LIN {X 0,Y 418.278,Z 217.377,A -85,B 0,C 180,E1 -10094.598,E2 -10094.598} C_VEL
LIN {X 0,Y 418.254,Z 217.38,A -85,B 0,C 180,E1 -10097.606,E2 -10097.606} C_VEL
LIN {X 0,Y 418.225,Z 217.388,A -85,B 0,C 180,E1 -10100.665,E2 -10100.665} C_VEL
LIN {X 0,Y 418.244,Z 217.38,A -85,B 0,C 180,E1 -10103.784,E2 -10103.784} C_VEL
LIN {X 0,Y 418.204,Z 217.387,A -85,B 0,C 180,E1 -10107.049,E2 -10107.049} C_VEL
LIN {X 0,Y 418.221,Z 217.39,A -85,B 0,C 180,E1 -10110.274,E2 -10110.274} C_VEL
LIN {X 0,Y 418.215,Z 217.387,A -85,B 0,C 180,E1 -10113.681,E2 -10113.681} C_VEL
LIN {X 0,Y 418.222,Z 217.384,A -85,B 0,C 180,E1 -10117.226,E2 -10117.226} C_VEL
LIN {X 0,Y 418.217,Z 217.389,A -85,B 0,C 180,E1 -10119.686,E2 -10119.686} C_VEL
LIN {X 0,Y 418.211,Z 217.381,A -85,B 0,C 180,E1 -10122.322,E2 -10122.322} C_VEL
LIN {X 0,Y 418.224,Z 217.386,A -85,B 0,C 180,E1 -10125.11,E2 -10125.11} C_VEL
LIN {X 0,Y 418.223,Z 217.388,A -85,B 0,C 180,E1 -10127.767,E2 -10127.767} C_VEL
LIN {X 0,Y 418.231,Z 217.388,A -85,B 0,C 180,E1 -10131.558,E2 -10131.558} C_VEL
LIN {X 0,Y 418.255,Z 217.385,A -85,B 0,C 180,E1 -10135.16,E2 -10135.16} C_VEL
LIN {X 0,Y 418.242,Z 217.388,A -85,B 0,C 180,E1 -10137.473,E2 -10137.473} C_VEL
LIN {X 0,Y 418.296,Z 217.38,A -85,B 0,C 180,E1 -10141.146,E2 -10141.146} C_VEL
LIN {X 0,Y 418.289,Z 217.454,A -85,B 0,C 180,E1 -10141.329,E2 -10141.329} C_VEL
LIN {X 0,Y 421.211,Z 231.065,A -85,B 0,C 180,E1 -10144.291,E2 -10144.291} C_VEL
LIN {X 0,Y 421.805,Z 235.075,A -85,B 0,C 180,E1 -10145.121,E2 -10145.121} C_VEL
LIN {X 0,Y 420.665,Z 251.075,A -85,B 0,C 180,E1 -10148.178,E2 -10148.178} C_VEL
LIN {X 0,Y 419.91,Z 263.661,A -85,B 0,C 180,E1 -10150.553,E2 -10150.553} C_VEL
LIN {X 0,Y 423.793,Z 286.997,A -85,B 0,C 180,E1 -10151.184,E2 -10151.184} C_VEL
LIN {X 0,Y 424.441,Z 292.599,A -85,B 0,C 180,E1 -10151.319,E2 -10151.319} C_VEL
LIN {X 0,Y 423.429,Z 373.284,A -85,B 0,C 180,E1 -10152.741,E2 -10152.741} C_VEL
LIN {X 0,Y 422.9,Z 386.195,A -85,B 0,C 180,E1 -10153.155,E2 -10153.155} C_VEL
LIN {X 0,Y 422.122,Z 398.74,A -85,B 0,C 180,E1 -10153.745,E2 -10153.745} C_VEL
LIN {X 0,Y 421.283,Z 410.718,A -85,B 0,C 180,E1 -10154.519,E2 -10154.519} C_VEL
LIN {X 0,Y 420.456,Z 422.181,A -85,B 0,C 180,E1 -10155.479,E2 -10155.479} C_VEL
LIN {X 0,Y 419.612,Z 432.537,A -85,B 0,C 180,E1 -10156.562,E2 -10156.562} C_VEL
LIN {X 0,Y 419.023,Z 441.025,A -85,B 0,C 180,E1 -10157.652,E2 -10157.652} C_VEL
LIN {X 0,Y 418.225,Z 450.262,A -85,B 0,C 180,E1 -10159.102,E2 -10159.102} C_VEL
LIN {X 0,Y 417.725,Z 457.708,A -85,B 0,C 180,E1 -10160.558,E2 -10160.558} C_VEL
LIN {X 0,Y 417.326,Z 464.595,A -85,B 0,C 180,E1 -10162.256,E2 -10162.256} C_VEL
LIN {X 0,Y 417.128,Z 469.27,A -85,B 0,C 180,E1 -10163.756,E2 -10163.756} C_VEL
LIN {X 0,Y 417.104,Z 472.633,A -85,B 0,C 180,E1 -10165.166,E2 -10165.166} C_VEL
LIN {X 0,Y 417.07,Z 475.706,A -85,B 0,C 180,E1 -10167.101,E2 -10167.101} C_VEL
LIN {X 0,Y 417.091,Z 476.646,A -85,B 0,C 180,E1 -10168.067,E2 -10168.067} C_VEL
LIN {X 0,Y 417.058,Z 477.181,A -85,B 0,C 180,E1 -10169.033,E2 -10169.033} C_VEL
LIN {X 0,Y 417.057,Z 477.284,A -85,B 0,C 180,E1 -10169.998,E2 -10169.998} C_VEL
LIN {X 0,Y 417.091,Z 476.323,A -85,B 0,C 180,E1 -10171.929,E2 -10171.929} C_VEL
LIN {X 0,Y 417.088,Z 475.245,A -85,B 0,C 180,E1 -10172.896,E2 -10172.896} C_VEL
LIN {X 0,Y 417.023,Z 473.703,A -85,B 0,C 180,E1 -10173.863,E2 -10173.863} C_VEL
LIN {X 0,Y 417.13,Z 470.604,A -85,B 0,C 180,E1 -10175.315,E2 -10175.315} C_VEL
LIN {X 0,Y 417.229,Z 466.427,A -85,B 0,C 180,E1 -10176.769,E2 -10176.769} C_VEL
LIN {X 0,Y 417.451,Z 460.038,A -85,B 0,C 180,E1 -10178.469,E2 -10178.469} C_VEL
LIN {X 0,Y 417.799,Z 453.074,A -85,B 0,C 180,E1 -10179.926,E2 -10179.926} C_VEL
LIN {X 0,Y 418.316,Z 444.342,A -85,B 0,C 180,E1 -10181.383,E2 -10181.383} C_VEL
LIN {X 0,Y 418.877,Z 435.383,A -85,B 0,C 180,E1 -10182.596,E2 -10182.596} C_VEL
LIN {X 0,Y 419.619,Z 424.593,A -85,B 0,C 180,E1 -10183.78,E2 -10183.78} C_VEL
LIN {X 0,Y 420.27,Z 413.141,A -85,B 0,C 180,E1 -10184.772,E2 -10184.772} C_VEL
LIN {X 0,Y 421.02,Z 400.592,A -85,B 0,C 180,E1 -10185.612,E2 -10185.612} C_VEL
LIN {X 0,Y 421.634,Z 387.804,A -85,B 0,C 180,E1 -10186.24,E2 -10186.24} C_VEL
LIN {X 0,Y 422.161,Z 374.192,A -85,B 0,C 180,E1 -10186.685,E2 -10186.685} C_VEL
LIN {X 0,Y 422.539,Z 344.069,A -85,B 0,C 180,E1 -10187.23,E2 -10187.23} C_VEL
LIN {X 0,Y 422.928,Z 289.758,A -85,B 0,C 180,E1 -10188.161,E2 -10188.161} C_VEL
LIN {X 0,Y 419.318,Z 264.152,A -85,B 0,C 180,E1 -10188.756,E2 -10188.756} C_VEL
LIN {X 0,Y 420.39,Z 244.757,A -85,B 0,C 180,E1 -10192.35,E2 -10192.35} C_VEL
LIN {X 0,Y 421.057,Z 232.437,A -85,B 0,C 180,E1 -10194.659,E2 -10194.659} C_VEL
LIN {X 0,Y 419.409,Z 222.603,A -85,B 0,C 180,E1 -10196.627,E2 -10196.627} C_VEL
LIN {X 0,Y 418.358,Z 217.376,A -85,B 0,C 180,E1 -10197.726,E2 -10197.726} C_VEL
LIN {X 0,Y 418.196,Z 217.389,A -85,B 0,C 180,E1 -10201.392,E2 -10201.392} C_VEL
LIN {X 0,Y 418.248,Z 217.384,A -85,B 0,C 180,E1 -10204.576,E2 -10204.576} C_VEL
LIN {X 0,Y 418.208,Z 217.393,A -85,B 0,C 180,E1 -10207.829,E2 -10207.829} C_VEL
LIN {X 0,Y 418.199,Z 217.388,A -85,B 0,C 180,E1 -10210.944,E2 -10210.944} C_VEL
LIN {X 0,Y 418.185,Z 217.396,A -85,B 0,C 180,E1 -10213.725,E2 -10213.725} C_VEL
LIN {X 0,Y 418.234,Z 217.385,A -85,B 0,C 180,E1 -10216.451,E2 -10216.451} C_VEL
LIN {X 0,Y 418.238,Z 217.384,A -85,B 0,C 180,E1 -10219.119,E2 -10219.119} C_VEL
LIN {X 0,Y 418.206,Z 217.39,A -85,B 0,C 180,E1 -10222.161,E2 -10222.161} C_VEL
LIN {X 0,Y 418.23,Z 217.389,A -85,B 0,C 180,E1 -10225.416,E2 -10225.416} C_VEL
LIN {X 0,Y 418.177,Z 217.391,A -85,B 0,C 180,E1 -10228.601,E2 -10228.601} C_VEL
LIN {X 0,Y 418.255,Z 217.384,A -85,B 0,C 180,E1 -10231.934,E2 -10231.934} C_VEL
LIN {X 0,Y 418.249,Z 217.385,A -85,B 0,C 180,E1 -10235.16,E2 -10235.16} C_VEL
LIN {X 0,Y 418.218,Z 217.386,A -85,B 0,C 180,E1 -10238.302,E2 -10238.302} C_VEL
LIN {X 0,Y 418.239,Z 217.391,A -85,B 0,C 180,E1 -10241.381,E2 -10241.381} C_VEL
LIN {X 0,Y 418.263,Z 217.38,A -85,B 0,C 180,E1 -10244.404,E2 -10244.404} C_VEL
LIN {X 0,Y 418.323,Z 217.379,A -85,B 0,C 180,E1 -10247.384,E2 -10247.384} C_VEL
LIN {X 0,Y 418.368,Z 217.374,A -85,B 0,C 180,E1 -10251.304,E2 -10251.304} C_VEL
LIN {X 0,Y 418.49,Z 217.352,A -85,B 0,C 180,E1 -10254.217,E2 -10254.217} C_VEL
LIN {X 0,Y 418.492,Z 217.352,A -85,B 0,C 180,E1 -10258.075,E2 -10258.075} C_VEL
LIN {X 0,Y 418.62,Z 217.336,A -85,B 0,C 180,E1 -10260,E2 -10260} C_VEL
LIN {X 0,Y 418.45,Z 217.363,A -85,B 0,C 180,E1 -10262.888,E2 -10262.888} C_VEL
LIN {X 0,Y 418.438,Z 217.363,A -85,B 0,C 180,E1 -10266.752,E2 -10266.752} C_VEL
LIN {X 0,Y 418.294,Z 217.377,A -85,B 0,C 180,E1 -10269.672,E2 -10269.672} C_VEL
LIN {X 0,Y 418.306,Z 217.38,A -85,B 0,C 180,E1 -10273.007,E2 -10273.007} C_VEL
LIN {X 0,Y 418.272,Z 217.386,A -85,B 0,C 180,E1 -10276.74,E2 -10276.74} C_VEL
LIN {X 0,Y 418.223,Z 217.385,A -85,B 0,C 180,E1 -10279.791,E2 -10279.791} C_VEL
LIN {X 0,Y 418.187,Z 217.397,A -85,B 0,C 180,E1 -10282.739,E2 -10282.739} C_VEL
LIN {X 0,Y 418.226,Z 217.385,A -85,B 0,C 180,E1 -10285.907,E2 -10285.907} C_VEL
LIN {X 0,Y 418.223,Z 217.386,A -85,B 0,C 180,E1 -10289.165,E2 -10289.165} C_VEL
LIN {X 0,Y 418.218,Z 217.389,A -85,B 0,C 180,E1 -10292.847,E2 -10292.847} C_VEL
LIN {X 0,Y 418.208,Z 217.392,A -85,B 0,C 180,E1 -10296.241,E2 -10296.241} C_VEL
LIN {X 0,Y 418.208,Z 217.388,A -85,B 0,C 180,E1 -10299.686,E2 -10299.686} C_VEL
LIN {X 0,Y 418.196,Z 217.396,A -85,B 0,C 180,E1 -10302.324,E2 -10302.324} C_VEL
LIN {X 0,Y 418.205,Z 217.388,A -85,B 0,C 180,E1 -10305.112,E2 -10305.112} C_VEL
LIN {X 0,Y 418.212,Z 217.389,A -85,B 0,C 180,E1 -10307.77,E2 -10307.77} C_VEL
LIN {X 0,Y 418.232,Z 217.387,A -85,B 0,C 180,E1 -10310.622,E2 -10310.622} C_VEL
LIN {X 0,Y 418.221,Z 217.391,A -85,B 0,C 180,E1 -10313.98,E2 -10313.98} C_VEL
LIN {X 0,Y 418.238,Z 217.383,A -85,B 0,C 180,E1 -10317.16,E2 -10317.16} C_VEL
LIN {X 0,Y 418.252,Z 217.382,A -85,B 0,C 180,E1 -10320.899,E2 -10320.899} C_VEL
LIN {X 0,Y 418.254,Z 217.387,A -85,B 0,C 180,E1 -10324.099,E2 -10324.099} C_VEL
LIN {X 0,Y 418.22,Z 217.386,A -85,B 0,C 180,E1 -10327.267,E2 -10327.267} C_VEL
LIN {X 0,Y 418.273,Z 217.381,A -85,B 0,C 180,E1 -10330.367,E2 -10330.367} C_VEL
LIN {X 0,Y 418.308,Z 217.377,A -85,B 0,C 180,E1 -10333.408,E2 -10333.408} C_VEL
LIN {X 0,Y 418.34,Z 217.371,A -85,B 0,C 180,E1 -10337.002,E2 -10337.002} C_VEL
LIN {X 0,Y 418.334,Z 217.372,A -85,B 0,C 180,E1 -10340.331,E2 -10340.331} C_VEL
LIN {X 0,Y 418.456,Z 217.363,A -85,B 0,C 180,E1 -10343.251,E2 -10343.251} C_VEL
LIN {X 0,Y 418.477,Z 217.455,A -85,B 0,C 180,E1 -10343.947,E2 -10343.947} C_VEL
LIN {X 0,Y 419.779,Z 226.103,A -85,B 0,C 180,E1 -10345.922,E2 -10345.922} C_VEL
LIN {X 0,Y 419.767,Z 228.219,A -85,B 0,C 180,E1 -10346.357,E2 -10346.357} C_VEL
LIN {X 0,Y 423.446,Z 246.784,A -85,B 0,C 180,E1 -10346.827,E2 -10346.827} C_VEL
LIN {X 0,Y 422.508,Z 326.828,A -85,B 0,C 180,E1 -10348.186,E2 -10348.186} C_VEL
LIN {X 0,Y 421.787,Z 330.749,A -85,B 0,C 180,E1 -10348.232,E2 -10348.232} C_VEL
LIN {X 0,Y 415.99,Z 342.937,A -85,B 0,C 180,E1 -10348.344,E2 -10348.344} C_VEL
LIN {X 0,Y 415.247,Z 346.753,A -85,B 0,C 180,E1 -10348.46,E2 -10348.46} C_VEL
LIN {X 0,Y 414.843,Z 359.25,A -85,B 0,C 180,E1 -10349.031,E2 -10349.031} C_VEL
LIN {X 0,Y 414.324,Z 370.985,A -85,B 0,C 180,E1 -10349.758,E2 -10349.758} C_VEL
LIN {X 0,Y 413.654,Z 381.718,A -85,B 0,C 180,E1 -10350.61,E2 -10350.61} C_VEL
LIN {X 0,Y 412.91,Z 392.654,A -85,B 0,C 180,E1 -10351.708,E2 -10351.708} C_VEL
LIN {X 0,Y 412.267,Z 402.428,A -85,B 0,C 180,E1 -10352.933,E2 -10352.933} C_VEL
LIN {X 0,Y 411.654,Z 410.465,A -85,B 0,C 180,E1 -10354.162,E2 -10354.162} C_VEL
LIN {X 0,Y 411.105,Z 418.344,A -85,B 0,C 180,E1 -10355.642,E2 -10355.642} C_VEL
LIN {X 0,Y 410.777,Z 424.544,A -85,B 0,C 180,E1 -10357.106,E2 -10357.106} C_VEL
LIN {X 0,Y 410.393,Z 430.353,A -85,B 0,C 180,E1 -10358.867,E2 -10358.867} C_VEL
LIN {X 0,Y 410.172,Z 434.052,A -85,B 0,C 180,E1 -10360.365,E2 -10360.365} C_VEL
LIN {X 0,Y 410.037,Z 437.334,A -85,B 0,C 180,E1 -10362.32,E2 -10362.32} C_VEL
LIN {X 0,Y 409.887,Z 438.786,A -85,B 0,C 180,E1 -10363.89,E2 -10363.89} C_VEL
LIN {X 0,Y 409.889,Z 439.171,A -85,B 0,C 180,E1 -10364.904,E2 -10364.904} C_VEL
LIN {X 0,Y 409.922,Z 439.074,A -85,B 0,C 180,E1 -10366.24,E2 -10366.24} C_VEL
LIN {X 0,Y 409.98,Z 437.835,A -85,B 0,C 180,E1 -10367.973,E2 -10367.973} C_VEL
LIN {X 0,Y 410.24,Z 435.587,A -85,B 0,C 180,E1 -10369.572,E2 -10369.572} C_VEL
LIN {X 0,Y 410.472,Z 432.468,A -85,B 0,C 180,E1 -10371.073,E2 -10371.073} C_VEL
LIN {X 0,Y 410.829,Z 427.769,A -85,B 0,C 180,E1 -10372.731,E2 -10372.731} C_VEL
LIN {X 0,Y 411.322,Z 422.338,A -85,B 0,C 180,E1 -10374.209,E2 -10374.209} C_VEL
LIN {X 0,Y 411.979,Z 415.054,A -85,B 0,C 180,E1 -10375.785,E2 -10375.785} C_VEL
LIN {X 0,Y 412.672,Z 407.471,A -85,B 0,C 180,E1 -10377.1,E2 -10377.1} C_VEL
LIN {X 0,Y 413.52,Z 398.148,A -85,B 0,C 180,E1 -10378.415,E2 -10378.415} C_VEL
LIN {X 0,Y 414.375,Z 388.005,A -85,B 0,C 180,E1 -10379.574,E2 -10379.574} C_VEL
LIN {X 0,Y 415.205,Z 377.739,A -85,B 0,C 180,E1 -10380.516,E2 -10380.516} C_VEL
LIN {X 0,Y 415.907,Z 365.838,A -85,B 0,C 180,E1 -10381.376,E2 -10381.376} C_VEL
LIN {X 0,Y 416.547,Z 352.72,A -85,B 0,C 180,E1 -10382.084,E2 -10382.084} C_VEL
LIN {X 0,Y 416.978,Z 339.811,A -85,B 0,C 180,E1 -10382.558,E2 -10382.558} C_VEL
LIN {X 0,Y 417.233,Z 323.651,A -85,B 0,C 180,E1 -10382.902,E2 -10382.902} C_VEL
LIN {X 0,Y 418.307,Z 248.25,A -85,B 0,C 180,E1 -10384.226,E2 -10384.226} C_VEL
LIN {X 0,Y 414.744,Z 232.783,A -85,B 0,C 180,E1 -10384.718,E2 -10384.718} C_VEL
LIN {X 0,Y 413.422,Z 228.606,A -85,B 0,C 180,E1 -10384.897,E2 -10384.897} C_VEL
LIN {X 0,Y 411.214,Z 218.263,A -85,B 0,C 180,E1 -10387.428,E2 -10387.428} C_VEL
LIN {X 0,Y 411.203,Z 218.265,A -85,B 0,C 180,E1 -10390.499,E2 -10390.499} C_VEL
LIN {X 0,Y 411.211,Z 218.265,A -85,B 0,C 180,E1 -10393.126,E2 -10393.126} C_VEL
LIN {X 0,Y 411.227,Z 218.261,A -85,B 0,C 180,E1 -10395.87,E2 -10395.87} C_VEL
LIN {X 0,Y 411.197,Z 218.264,A -85,B 0,C 180,E1 -10399.498,E2 -10399.498} C_VEL
LIN {X 0,Y 411.187,Z 218.265,A -85,B 0,C 180,E1 -10402.026,E2 -10402.026} C_VEL
LIN {X 0,Y 411.188,Z 218.262,A -85,B 0,C 180,E1 -10405.665,E2 -10405.665} C_VEL
LIN {X 0,Y 411.177,Z 218.262,A -85,B 0,C 180,E1 -10409.152,E2 -10409.152} C_VEL
LIN {X 0,Y 411.24,Z 218.255,A -85,B 0,C 180,E1 -10412.521,E2 -10412.521} C_VEL
LIN {X 0,Y 411.207,Z 218.259,A -85,B 0,C 180,E1 -10415.784,E2 -10415.784} C_VEL
LIN {X 0,Y 411.196,Z 218.256,A -85,B 0,C 180,E1 -10418.966,E2 -10418.966} C_VEL
LIN {X 0,Y 411.229,Z 218.255,A -85,B 0,C 180,E1 -10422.084,E2 -10422.084} C_VEL
LIN {X 0,Y 411.238,Z 218.258,A -85,B 0,C 180,E1 -10425.147,E2 -10425.147} C_VEL
LIN {X 0,Y 411.257,Z 218.253,A -85,B 0,C 180,E1 -10428.167,E2 -10428.167} C_VEL
LIN {X 0,Y 411.419,Z 218.228,A -85,B 0,C 180,E1 -10432.186,E2 -10432.186} C_VEL
LIN {X 0,Y 411.452,Z 218.229,A -85,B 0,C 180,E1 -10434.118,E2 -10434.118} C_VEL
LIN {X 0,Y 411.481,Z 218.223,A -85,B 0,C 180,E1 -10438.043,E2 -10438.043} C_VEL
LIN {X 0,Y 411.611,Z 218.205,A -85,B 0,C 180,E1 -10440,E2 -10440} C_VEL
LIN {X 0,Y 411.428,Z 218.231,A -85,B 0,C 180,E1 -10442.938,E2 -10442.938} C_VEL
LIN {X 0,Y 411.404,Z 218.231,A -85,B 0,C 180,E1 -10446.868,E2 -10446.868} C_VEL
LIN {X 0,Y 411.269,Z 218.244,A -85,B 0,C 180,E1 -10449.84,E2 -10449.84} C_VEL
LIN {X 0,Y 411.289,Z 218.25,A -85,B 0,C 180,E1 -10453.109,E2 -10453.109} C_VEL
LIN {X 0,Y 411.245,Z 218.26,A -85,B 0,C 180,E1 -10456.89,E2 -10456.89} C_VEL
LIN {X 0,Y 411.188,Z 218.259,A -85,B 0,C 180,E1 -10459.989,E2 -10459.989} C_VEL
LIN {X 0,Y 411.17,Z 218.263,A -85,B 0,C 180,E1 -10463.15,E2 -10463.15} C_VEL
LIN {X 0,Y 411.166,Z 218.269,A -85,B 0,C 180,E1 -10466.386,E2 -10466.386} C_VEL
LIN {X 0,Y 411.178,Z 218.264,A -85,B 0,C 180,E1 -10469.715,E2 -10469.715} C_VEL
LIN {X 0,Y 411.188,Z 218.263,A -85,B 0,C 180,E1 -10473.158,E2 -10473.158} C_VEL
LIN {X 0,Y 411.176,Z 218.268,A -85,B 0,C 180,E1 -10476.554,E2 -10476.554} C_VEL
LIN {X 0,Y 411.184,Z 218.265,A -85,B 0,C 180,E1 -10479.726,E2 -10479.726} C_VEL
LIN {X 0,Y 411.159,Z 218.266,A -85,B 0,C 180,E1 -10483.136,E2 -10483.136} C_VEL
LIN {X 0,Y 411.157,Z 218.269,A -85,B 0,C 180,E1 -10485.883,E2 -10485.883} C_VEL
LIN {X 0,Y 411.144,Z 218.269,A -85,B 0,C 180,E1 -10488.775,E2 -10488.775} C_VEL
LIN {X 0,Y 411.18,Z 218.27,A -85,B 0,C 180,E1 -10492.027,E2 -10492.027} C_VEL
LIN {X 0,Y 411.202,Z 218.263,A -85,B 0,C 180,E1 -10495.668,E2 -10495.668} C_VEL
LIN {X 0,Y 411.187,Z 218.267,A -85,B 0,C 180,E1 -10499.153,E2 -10499.153} C_VEL
LIN {X 0,Y 411.245,Z 218.386,A -85,B 0,C 180,E1 -10500.991,E2 -10500.991} C_VEL
LIN {X 0,Y 414.024,Z 231.041,A -85,B 0,C 180,E1 -10503.811,E2 -10503.811} C_VEL
LIN {X 0,Y 414.931,Z 236.363,A -85,B 0,C 180,E1 -10504.948,E2 -10504.948} C_VEL
LIN {X 0,Y 413.75,Z 252.357,A -85,B 0,C 180,E1 -10508.057,E2 -10508.057} C_VEL
LIN {X 0,Y 413.073,Z 263.481,A -85,B 0,C 180,E1 -10510.165,E2 -10510.165} C_VEL
LIN {X 0,Y 417.131,Z 287.273,A -85,B 0,C 180,E1 -10510.834,E2 -10510.834} C_VEL
LIN {X 0,Y 417.841,Z 294.938,A -85,B 0,C 180,E1 -10511.012,E2 -10511.012} C_VEL
LIN {X 0,Y 416.762,Z 372.395,A -85,B 0,C 180,E1 -10512.393,E2 -10512.393} C_VEL
LIN {X 0,Y 416.204,Z 385.488,A -85,B 0,C 180,E1 -10512.812,E2 -10512.812} C_VEL
LIN {X 0,Y 415.417,Z 398.126,A -85,B 0,C 180,E1 -10513.412,E2 -10513.412} C_VEL
LIN {X 0,Y 414.576,Z 409.396,A -85,B 0,C 180,E1 -10514.136,E2 -10514.136} C_VEL
LIN {X 0,Y 413.676,Z 421.043,A -85,B 0,C 180,E1 -10515.11,E2 -10515.11} C_VEL
LIN {X 0,Y 412.805,Z 431.536,A -85,B 0,C 180,E1 -10516.21,E2 -10516.21} C_VEL
LIN {X 0,Y 412.073,Z 441.02,A -85,B 0,C 180,E1 -10517.44,E2 -10517.44} C_VEL
LIN {X 0,Y 411.243,Z 450.174,A -85,B 0,C 180,E1 -10518.915,E2 -10518.915} C_VEL
LIN {X 0,Y 410.699,Z 457.569,A -85,B 0,C 180,E1 -10520.395,E2 -10520.395} C_VEL
LIN {X 0,Y 410.268,Z 464.398,A -85,B 0,C 180,E1 -10522.122,E2 -10522.122} C_VEL
LIN {X 0,Y 410.044,Z 469.361,A -85,B 0,C 180,E1 -10523.775,E2 -10523.775} C_VEL
LIN {X 0,Y 410.011,Z 472.377,A -85,B 0,C 180,E1 -10525.082,E2 -10525.082} C_VEL
LIN {X 0,Y 409.967,Z 475.422,A -85,B 0,C 180,E1 -10527.051,E2 -10527.051} C_VEL
LIN {X 0,Y 410.018,Z 476.351,A -85,B 0,C 180,E1 -10528.034,E2 -10528.034} C_VEL
LIN {X 0,Y 409.981,Z 476.862,A -85,B 0,C 180,E1 -10529.016,E2 -10529.016} C_VEL
LIN {X 0,Y 409.976,Z 476.95,A -85,B 0,C 180,E1 -10529.998,E2 -10529.998} C_VEL
LIN {X 0,Y 410.019,Z 475.965,A -85,B 0,C 180,E1 -10531.963,E2 -10531.963} C_VEL
LIN {X 0,Y 409.987,Z 474.861,A -85,B 0,C 180,E1 -10532.946,E2 -10532.946} C_VEL
LIN {X 0,Y 409.942,Z 473.303,A -85,B 0,C 180,E1 -10533.93,E2 -10533.93} C_VEL
LIN {X 0,Y 410.025,Z 470.174,A -85,B 0,C 180,E1 -10535.407,E2 -10535.407} C_VEL
LIN {X 0,Y 410.16,Z 465.968,A -85,B 0,C 180,E1 -10536.886,E2 -10536.886} C_VEL
LIN {X 0,Y 410.378,Z 459.543,A -85,B 0,C 180,E1 -10538.616,E2 -10538.616} C_VEL
LIN {X 0,Y 410.737,Z 452.536,A -85,B 0,C 180,E1 -10540.098,E2 -10540.098} C_VEL
LIN {X 0,Y 411.306,Z 443.743,A -85,B 0,C 180,E1 -10541.579,E2 -10541.579} C_VEL
LIN {X 0,Y 411.921,Z 434.723,A -85,B 0,C 180,E1 -10542.812,E2 -10542.812} C_VEL
LIN {X 0,Y 412.602,Z 424.803,A -85,B 0,C 180,E1 -10543.919,E2 -10543.919} C_VEL
LIN {X 0,Y 413.277,Z 413.842,A -85,B 0,C 180,E1 -10544.901,E2 -10544.901} C_VEL
LIN {X 0,Y 414.015,Z 401.537,A -85,B 0,C 180,E1 -10545.756,E2 -10545.756} C_VEL
LIN {X 0,Y 414.68,Z 388.616,A -85,B 0,C 180,E1 -10546.425,E2 -10546.425} C_VEL
LIN {X 0,Y 415.212,Z 375.583,A -85,B 0,C 180,E1 -10546.878,E2 -10546.878} C_VEL
LIN {X 0,Y 415.506,Z 358.931,A -85,B 0,C 180,E1 -10547.214,E2 -10547.214} C_VEL
LIN {X 0,Y 416.104,Z 290.614,A -85,B 0,C 180,E1 -10548.4,E2 -10548.4} C_VEL
LIN {X 0,Y 412.373,Z 263.746,A -85,B 0,C 180,E1 -10549.051,E2 -10549.051} C_VEL
LIN {X 0,Y 413.58,Z 242.792,A -85,B 0,C 180,E1 -10553.003,E2 -10553.003} C_VEL
LIN {X 0,Y 414.076,Z 233.186,A -85,B 0,C 180,E1 -10554.835,E2 -10554.835} C_VEL
LIN {X 0,Y 411.933,Z 221.274,A -85,B 0,C 180,E1 -10557.277,E2 -10557.277} C_VEL
LIN {X 0,Y 411.296,Z 218.257,A -85,B 0,C 180,E1 -10557.954,E2 -10557.954} C_VEL
LIN {X 0,Y 411.168,Z 218.264,A -85,B 0,C 180,E1 -10561.279,E2 -10561.279} C_VEL
LIN {X 0,Y 411.189,Z 218.265,A -85,B 0,C 180,E1 -10564.329,E2 -10564.329} C_VEL
LIN {X 0,Y 411.174,Z 218.271,A -85,B 0,C 180,E1 -10567.97,E2 -10567.97} C_VEL
LIN {X 0,Y 411.14,Z 218.268,A -85,B 0,C 180,E1 -10571.224,E2 -10571.224} C_VEL
LIN {X 0,Y 411.155,Z 218.267,A -85,B 0,C 180,E1 -10574.486,E2 -10574.486} C_VEL
LIN {X 0,Y 411.199,Z 218.262,A -85,B 0,C 180,E1 -10577.293,E2 -10577.293} C_VEL
LIN {X 0,Y 411.201,Z 218.26,A -85,B 0,C 180,E1 -10580.774,E2 -10580.774} C_VEL
LIN {X 0,Y 411.165,Z 218.265,A -85,B 0,C 180,E1 -10584.468,E2 -10584.468} C_VEL
LIN {X 0,Y 411.172,Z 218.264,A -85,B 0,C 180,E1 -10586.87,E2 -10586.87} C_VEL
LIN {X 0,Y 411.201,Z 218.26,A -85,B 0,C 180,E1 -10590.639,E2 -10590.639} C_VEL
LIN {X 0,Y 411.199,Z 218.266,A -85,B 0,C 180,E1 -10593.616,E2 -10593.616} C_VEL
LIN {X 0,Y 411.214,Z 218.264,A -85,B 0,C 180,E1 -10597.337,E2 -10597.337} C_VEL
LIN {X 0,Y 411.222,Z 218.258,A -85,B 0,C 180,E1 -10600.029,E2 -10600.029} C_VEL
LIN {X 0,Y 411.219,Z 218.262,A -85,B 0,C 180,E1 -10603.129,E2 -10603.129} C_VEL
LIN {X 0,Y 411.266,Z 218.254,A -85,B 0,C 180,E1 -10606.89,E2 -10606.89} C_VEL
LIN {X 0,Y 411.265,Z 218.252,A -85,B 0,C 180,E1 -10610.16,E2 -10610.16} C_VEL
LIN {X 0,Y 411.429,Z 218.238,A -85,B 0,C 180,E1 -10613.132,E2 -10613.132} C_VEL
LIN {X 0,Y 411.268,Z 218.258,A -85,B 0,C 180,E1 -10615.098,E2 -10615.098} C_VEL
LIN {X 0,Y 411.461,Z 218.228,A -85,B 0,C 180,E1 -10618.042,E2 -10618.042} C_VEL
LIN {X 0,Y 411.59,Z 218.212,A -85,B 0,C 180,E1 -10620,E2 -10620} C_VEL
LIN {X 0,Y 411.407,Z 218.241,A -85,B 0,C 180,E1 -10622.937,E2 -10622.937} C_VEL
LIN {X 0,Y 411.402,Z 218.241,A -85,B 0,C 180,E1 -10626.868,E2 -10626.868} C_VEL
LIN {X 0,Y 411.247,Z 218.254,A -85,B 0,C 180,E1 -10629.84,E2 -10629.84} C_VEL
LIN {X 0,Y 411.265,Z 218.256,A -85,B 0,C 180,E1 -10633.109,E2 -10633.109} C_VEL
LIN {X 0,Y 411.215,Z 218.264,A -85,B 0,C 180,E1 -10636.89,E2 -10636.89} C_VEL
LIN {X 0,Y 411.164,Z 218.265,A -85,B 0,C 180,E1 -10639.99,E2 -10639.99} C_VEL
LIN {X 0,Y 411.152,Z 218.268,A -85,B 0,C 180,E1 -10643.15,E2 -10643.15} C_VEL
LIN {X 0,Y 411.195,Z 218.265,A -85,B 0,C 180,E1 -10646.384,E2 -10646.384} C_VEL
LIN {X 0,Y 411.159,Z 218.265,A -85,B 0,C 180,E1 -10649.716,E2 -10649.716} C_VEL
LIN {X 0,Y 411.168,Z 218.265,A -85,B 0,C 180,E1 -10653.159,E2 -10653.159} C_VEL
LIN {X 0,Y 411.156,Z 218.272,A -85,B 0,C 180,E1 -10656.556,E2 -10656.556} C_VEL
LIN {X 0,Y 411.173,Z 218.264,A -85,B 0,C 180,E1 -10659.73,E2 -10659.73} C_VEL
LIN {X 0,Y 411.141,Z 218.268,A -85,B 0,C 180,E1 -10663.137,E2 -10663.137} C_VEL
LIN {X 0,Y 411.139,Z 218.27,A -85,B 0,C 180,E1 -10665.885,E2 -10665.885} C_VEL
LIN {X 0,Y 411.138,Z 218.269,A -85,B 0,C 180,E1 -10668.775,E2 -10668.775} C_VEL
LIN {X 0,Y 411.182,Z 218.265,A -85,B 0,C 180,E1 -10671.835,E2 -10671.835} C_VEL
LIN {X 0,Y 411.19,Z 218.261,A -85,B 0,C 180,E1 -10675.125,E2 -10675.125} C_VEL
LIN {X 0,Y 411.146,Z 218.273,A -85,B 0,C 180,E1 -10678.006,E2 -10678.006} C_VEL
LIN {X 0,Y 411.201,Z 218.261,A -85,B 0,C 180,E1 -10681.414,E2 -10681.414} C_VEL
LIN {X 0,Y 411.222,Z 218.26,A -85,B 0,C 180,E1 -10683.623,E2 -10683.623} C_VEL
LIN {X 0,Y 411.183,Z 218.262,A -85,B 0,C 180,E1 -10686.855,E2 -10686.855} C_VEL
LIN {X 0,Y 411.204,Z 218.265,A -85,B 0,C 180,E1 -10690.054,E2 -10690.054} C_VEL
LIN {X 0,Y 411.255,Z 218.254,A -85,B 0,C 180,E1 -10693.134,E2 -10693.134} C_VEL
LIN {X 0,Y 411.299,Z 218.248,A -85,B 0,C 180,E1 -10696.899,E2 -10696.899} C_VEL
LIN {X 0,Y 411.286,Z 218.252,A -85,B 0,C 180,E1 -10700.164,E2 -10700.164} C_VEL
LIN {X 0,Y 411.42,Z 218.239,A -85,B 0,C 180,E1 -10703.135,E2 -10703.135} C_VEL
LIN {X 0,Y 411.42,Z 218.273,A -85,B 0,C 180,E1 -10703.75,E2 -10703.75} C_VEL
LIN {X 0,Y 412.817,Z 227.357,A -85,B 0,C 180,E1 -10705.853,E2 -10705.853} C_VEL
LIN {X 0,Y 412.784,Z 228.329,A -85,B 0,C 180,E1 -10706.066,E2 -10706.066} C_VEL
LIN {X 0,Y 416.633,Z 248.07,A -85,B 0,C 180,E1 -10706.584,E2 -10706.584} C_VEL
LIN {X 0,Y 415.517,Z 335.676,A -85,B 0,C 180,E1 -10708.117,E2 -10708.117} C_VEL
LIN {X 0,Y 415.247,Z 346.753,A -85,B 0,C 180,E1 -10708.46,E2 -10708.46} C_VEL
LIN {X 0,Y 414.791,Z 350.532,A -85,B 0,C 180,E1 -10708.599,E2 -10708.599} C_VEL
LIN {X 0,Y 412.675,Z 357.887,A -85,B 0,C 180,E1 -10708.878,E2 -10708.878} C_VEL
LIN {X 0,Y 408.624,Z 368.519,A -85,B 0,C 180,E1 -10709.384,E2 -10709.384} C_VEL
LIN {X 0,Y 407.341,Z 373.768,A -85,B 0,C 180,E1 -10709.725,E2 -10709.725} C_VEL
LIN {X 0,Y 407.152,Z 375.467,A -85,B 0,C 180,E1 -10709.856,E2 -10709.856} C_VEL
LIN {X 0,Y 406.374,Z 386.883,A -85,B 0,C 180,E1 -10710.869,E2 -10710.869} C_VEL
LIN {X 0,Y 405.664,Z 396.876,A -85,B 0,C 180,E1 -10711.987,E2 -10711.987} C_VEL
LIN {X 0,Y 405.016,Z 405.922,A -85,B 0,C 180,E1 -10713.234,E2 -10713.234} C_VEL
LIN {X 0,Y 404.404,Z 414.749,A -85,B 0,C 180,E1 -10714.736,E2 -10714.736} C_VEL
LIN {X 0,Y 403.901,Z 421.836,A -85,B 0,C 180,E1 -10716.245,E2 -10716.245} C_VEL
LIN {X 0,Y 403.479,Z 428.302,A -85,B 0,C 180,E1 -10718.011,E2 -10718.011} C_VEL
LIN {X 0,Y 403.189,Z 432.576,A -85,B 0,C 180,E1 -10719.533,E2 -10719.533} C_VEL
LIN {X 0,Y 403.035,Z 435.77,A -85,B 0,C 180,E1 -10721.059,E2 -10721.059} C_VEL
LIN {X 0,Y 402.939,Z 437.731,A -85,B 0,C 180,E1 -10722.383,E2 -10722.383} C_VEL
LIN {X 0,Y 402.804,Z 439.221,A -85,B 0,C 180,E1 -10724.139,E2 -10724.139} C_VEL
LIN {X 0,Y 402.806,Z 439.538,A -85,B 0,C 180,E1 -10725.172,E2 -10725.172} C_VEL
LIN {X 0,Y 402.837,Z 439.382,A -85,B 0,C 180,E1 -10726.354,E2 -10726.354} C_VEL
LIN {X 0,Y 402.933,Z 437.916,A -85,B 0,C 180,E1 -10728.298,E2 -10728.298} C_VEL
LIN {X 0,Y 403.181,Z 435.861,A -85,B 0,C 180,E1 -10729.731,E2 -10729.731} C_VEL
LIN {X 0,Y 403.468,Z 432.239,A -85,B 0,C 180,E1 -10731.457,E2 -10731.457} C_VEL
LIN {X 0,Y 403.893,Z 427.568,A -85,B 0,C 180,E1 -10733.08,E2 -10733.08} C_VEL
LIN {X 0,Y 404.439,Z 421.741,A -85,B 0,C 180,E1 -10734.648,E2 -10734.648} C_VEL
LIN {X 0,Y 405.197,Z 414.151,A -85,B 0,C 180,E1 -10736.249,E2 -10736.249} C_VEL
LIN {X 0,Y 405.944,Z 406.31,A -85,B 0,C 180,E1 -10737.588,E2 -10737.588} C_VEL
LIN {X 0,Y 406.815,Z 396.685,A -85,B 0,C 180,E1 -10738.928,E2 -10738.928} C_VEL
LIN {X 0,Y 407.671,Z 387.16,A -85,B 0,C 180,E1 -10739.995,E2 -10739.995} C_VEL
LIN {X 0,Y 408.631,Z 375.193,A -85,B 0,C 180,E1 -10741.061,E2 -10741.061} C_VEL
LIN {X 0,Y 409.391,Z 363.647,A -85,B 0,C 180,E1 -10741.861,E2 -10741.861} C_VEL
LIN {X 0,Y 409.966,Z 351.271,A -85,B 0,C 180,E1 -10742.501,E2 -10742.501} C_VEL
LIN {X 0,Y 410.355,Z 337.734,A -85,B 0,C 180,E1 -10742.975,E2 -10742.975} C_VEL
LIN {X 0,Y 410.996,Z 299.806,A -85,B 0,C 180,E1 -10743.684,E2 -10743.684} C_VEL
LIN {X 0,Y 411.835,Z 249.631,A -85,B 0,C 180,E1 -10744.574,E2 -10744.574} C_VEL
LIN {X 0,Y 408.153,Z 234.005,A -85,B 0,C 180,E1 -10745.089,E2 -10745.089} C_VEL
LIN {X 0,Y 406.263,Z 228.932,A -85,B 0,C 180,E1 -10745.328,E2 -10745.328} C_VEL
LIN {X 0,Y 404.145,Z 219.145,A -85,B 0,C 180,E1 -10747.804,E2 -10747.804} C_VEL
LIN {X 0,Y 404.154,Z 219.137,A -85,B 0,C 180,E1 -10751.358,E2 -10751.358} C_VEL
LIN {X 0,Y 404.186,Z 219.142,A -85,B 0,C 180,E1 -10754.528,E2 -10754.528} C_VEL
LIN {X 0,Y 404.197,Z 219.135,A -85,B 0,C 180,E1 -10757.304,E2 -10757.304} C_VEL
LIN {X 0,Y 404.155,Z 219.141,A -85,B 0,C 180,E1 -10759.954,E2 -10759.954} C_VEL
LIN {X 0,Y 404.124,Z 219.142,A -85,B 0,C 180,E1 -10763.123,E2 -10763.123} C_VEL
LIN {X 0,Y 404.127,Z 219.147,A -85,B 0,C 180,E1 -10766.186,E2 -10766.186} C_VEL
LIN {X 0,Y 404.133,Z 219.144,A -85,B 0,C 180,E1 -10769.714,E2 -10769.714} C_VEL
LIN {X 0,Y 404.175,Z 219.135,A -85,B 0,C 180,E1 -10773.122,E2 -10773.122} C_VEL
LIN {X 0,Y 404.151,Z 219.139,A -85,B 0,C 180,E1 -10776.425,E2 -10776.425} C_VEL
LIN {X 0,Y 404.184,Z 219.136,A -85,B 0,C 180,E1 -10779.868,E2 -10779.868} C_VEL
LIN {X 0,Y 404.195,Z 219.13,A -85,B 0,C 180,E1 -10782.992,E2 -10782.992} C_VEL
LIN {X 0,Y 404.259,Z 219.125,A -85,B 0,C 180,E1 -10786.938,E2 -10786.938} C_VEL
LIN {X 0,Y 404.232,Z 219.13,A -85,B 0,C 180,E1 -10789.988,E2 -10789.988} C_VEL
LIN {X 0,Y 404.384,Z 219.107,A -85,B 0,C 180,E1 -10793.013,E2 -10793.013} C_VEL
LIN {X 0,Y 404.257,Z 219.128,A -85,B 0,C 180,E1 -10795.014,E2 -10795.014} C_VEL
LIN {X 0,Y 404.451,Z 219.099,A -85,B 0,C 180,E1 -10798.009,E2 -10798.009} C_VEL
LIN {X 0,Y 404.581,Z 219.08,A -85,B 0,C 180,E1 -10800,E2 -10800} C_VEL
LIN {X 0,Y 404.386,Z 219.109,A -85,B 0,C 180,E1 -10802.989,E2 -10802.989} C_VEL
LIN {X 0,Y 404.355,Z 219.11,A -85,B 0,C 180,E1 -10806.989,E2 -10806.989} C_VEL
LIN {X 0,Y 404.237,Z 219.124,A -85,B 0,C 180,E1 -10811.026,E2 -10811.026} C_VEL
LIN {X 0,Y 404.187,Z 219.13,A -85,B 0,C 180,E1 -10814.089,E2 -10814.089} C_VEL
LIN {X 0,Y 404.184,Z 219.136,A -85,B 0,C 180,E1 -10817.194,E2 -10817.194} C_VEL
LIN {X 0,Y 404.134,Z 219.14,A -85,B 0,C 180,E1 -10820.353,E2 -10820.353} C_VEL
LIN {X 0,Y 404.132,Z 219.138,A -85,B 0,C 180,E1 -10823.577,E2 -10823.577} C_VEL
LIN {X 0,Y 404.109,Z 219.143,A -85,B 0,C 180,E1 -10826.884,E2 -10826.884} C_VEL
LIN {X 0,Y 404.125,Z 219.146,A -85,B 0,C 180,E1 -10830.287,E2 -10830.287} C_VEL
LIN {X 0,Y 404.122,Z 219.143,A -85,B 0,C 180,E1 -10833.815,E2 -10833.815} C_VEL
LIN {X 0,Y 404.119,Z 219.143,A -85,B 0,C 180,E1 -10836.876,E2 -10836.876} C_VEL
LIN {X 0,Y 404.137,Z 219.144,A -85,B 0,C 180,E1 -10840.082,E2 -10840.082} C_VEL
LIN {X 0,Y 404.139,Z 219.141,A -85,B 0,C 180,E1 -10843.085,E2 -10843.085} C_VEL
LIN {X 0,Y 404.138,Z 219.143,A -85,B 0,C 180,E1 -10845.927,E2 -10845.927} C_VEL
LIN {X 0,Y 404.1,Z 219.148,A -85,B 0,C 180,E1 -10848.635,E2 -10848.635} C_VEL
LIN {X 0,Y 404.134,Z 219.144,A -85,B 0,C 180,E1 -10851.496,E2 -10851.496} C_VEL
LIN {X 0,Y 404.18,Z 219.139,A -85,B 0,C 180,E1 -10854.985,E2 -10854.985} C_VEL
LIN {X 0,Y 404.139,Z 219.145,A -85,B 0,C 180,E1 -10858.555,E2 -10858.555} C_VEL
LIN {X 0,Y 404.196,Z 219.213,A -85,B 0,C 180,E1 -10860.612,E2 -10860.612} C_VEL
LIN {X 0,Y 406.836,Z 231.026,A -85,B 0,C 180,E1 -10863.312,E2 -10863.312} C_VEL
LIN {X 0,Y 408.047,Z 237.678,A -85,B 0,C 180,E1 -10864.769,E2 -10864.769} C_VEL
LIN {X 0,Y 406.84,Z 253.642,A -85,B 0,C 180,E1 -10867.931,E2 -10867.931} C_VEL
LIN {X 0,Y 406.199,Z 263.14,A -85,B 0,C 180,E1 -10869.755,E2 -10869.755} C_VEL
LIN {X 0,Y 409.938,Z 284.035,A -85,B 0,C 180,E1 -10870.369,E2 -10870.369} C_VEL
LIN {X 0,Y 411.262,Z 294.737,A -85,B 0,C 180,E1 -10870.644,E2 -10870.644} C_VEL
LIN {X 0,Y 410.141,Z 371.606,A -85,B 0,C 180,E1 -10872.035,E2 -10872.035} C_VEL
LIN {X 0,Y 409.623,Z 384.077,A -85,B 0,C 180,E1 -10872.431,E2 -10872.431} C_VEL
LIN {X 0,Y 408.84,Z 396.418,A -85,B 0,C 180,E1 -10873.008,E2 -10873.008} C_VEL
LIN {X 0,Y 407.902,Z 408.004,A -85,B 0,C 180,E1 -10873.741,E2 -10873.741} C_VEL
LIN {X 0,Y 406.919,Z 419.905,A -85,B 0,C 180,E1 -10874.729,E2 -10874.729} C_VEL
LIN {X 0,Y 406.005,Z 430.472,A -85,B 0,C 180,E1 -10875.839,E2 -10875.839} C_VEL
LIN {X 0,Y 405.135,Z 441.004,A -85,B 0,C 180,E1 -10877.221,E2 -10877.221} C_VEL
LIN {X 0,Y 404.257,Z 450.096,A -85,B 0,C 180,E1 -10878.721,E2 -10878.721} C_VEL
LIN {X 0,Y 403.664,Z 457.447,A -85,B 0,C 180,E1 -10880.226,E2 -10880.226} C_VEL
LIN {X 0,Y 403.204,Z 464.218,A -85,B 0,C 180,E1 -10881.983,E2 -10881.983} C_VEL
LIN {X 0,Y 402.935,Z 469.55,A -85,B 0,C 180,E1 -10883.826,E2 -10883.826} C_VEL
LIN {X 0,Y 402.92,Z 472.128,A -85,B 0,C 180,E1 -10884.995,E2 -10884.995} C_VEL
LIN {X 0,Y 402.865,Z 475.142,A -85,B 0,C 180,E1 -10886.999,E2 -10886.999} C_VEL
LIN {X 0,Y 402.946,Z 476.058,A -85,B 0,C 180,E1 -10887.999,E2 -10887.999} C_VEL
LIN {X 0,Y 402.906,Z 476.541,A -85,B 0,C 180,E1 -10888.999,E2 -10888.999} C_VEL
LIN {X 0,Y 402.899,Z 476.616,A -85,B 0,C 180,E1 -10889.998,E2 -10889.998} C_VEL
LIN {X 0,Y 402.948,Z 475.604,A -85,B 0,C 180,E1 -10891.997,E2 -10891.997} C_VEL
LIN {X 0,Y 402.887,Z 474.47,A -85,B 0,C 180,E1 -10892.998,E2 -10892.998} C_VEL
LIN {X 0,Y 402.863,Z 472.898,A -85,B 0,C 180,E1 -10893.999,E2 -10893.999} C_VEL
LIN {X 0,Y 402.922,Z 469.735,A -85,B 0,C 180,E1 -10895.503,E2 -10895.503} C_VEL
LIN {X 0,Y 403.071,Z 465.493,A -85,B 0,C 180,E1 -10897.008,E2 -10897.008} C_VEL
LIN {X 0,Y 403.327,Z 459.029,A -85,B 0,C 180,E1 -10898.767,E2 -10898.767} C_VEL
LIN {X 0,Y 403.69,Z 451.959,A -85,B 0,C 180,E1 -10900.277,E2 -10900.277} C_VEL
LIN {X 0,Y 404.319,Z 443.099,A -85,B 0,C 180,E1 -10901.782,E2 -10901.782} C_VEL
LIN {X 0,Y 404.975,Z 434.017,A -85,B 0,C 180,E1 -10903.035,E2 -10903.035} C_VEL
LIN {X 0,Y 405.686,Z 424.017,A -85,B 0,C 180,E1 -10904.161,E2 -10904.161} C_VEL
LIN {X 0,Y 406.33,Z 412.891,A -85,B 0,C 180,E1 -10905.162,E2 -10905.162} C_VEL
LIN {X 0,Y 407.138,Z 400.433,A -85,B 0,C 180,E1 -10906.03,E2 -10906.03} C_VEL
LIN {X 0,Y 407.781,Z 388.601,A -85,B 0,C 180,E1 -10906.647,E2 -10906.647} C_VEL
LIN {X 0,Y 408.316,Z 375.767,A -85,B 0,C 180,E1 -10907.107,E2 -10907.107} C_VEL
LIN {X 0,Y 408.644,Z 359.413,A -85,B 0,C 180,E1 -10907.448,E2 -10907.448} C_VEL
LIN {X 0,Y 409.283,Z 291.586,A -85,B 0,C 180,E1 -10908.645,E2 -10908.645} C_VEL
LIN {X 0,Y 405.39,Z 263.562,A -85,B 0,C 180,E1 -10909.31,E2 -10909.31} C_VEL
LIN {X 0,Y 406.598,Z 243.538,A -85,B 0,C 180,E1 -10913.152,E2 -10913.152} C_VEL
LIN {X 0,Y 407.1,Z 235.311,A -85,B 0,C 180,E1 -10914.745,E2 -10914.745} C_VEL
LIN {X 0,Y 405.996,Z 227.923,A -85,B 0,C 180,E1 -10916.265,E2 -10916.265} C_VEL
LIN {X 0,Y 404.249,Z 219.134,A -85,B 0,C 180,E1 -10918.132,E2 -10918.132} C_VEL
LIN {X 0,Y 404.124,Z 219.143,A -85,B 0,C 180,E1 -10921.554,E2 -10921.554} C_VEL
LIN {X 0,Y 404.167,Z 219.136,A -85,B 0,C 180,E1 -10925.012,E2 -10925.012} C_VEL
LIN {X 0,Y 404.133,Z 219.141,A -85,B 0,C 180,E1 -10928.753,E2 -10928.753} C_VEL
LIN {X 0,Y 404.099,Z 219.148,A -85,B 0,C 180,E1 -10931.595,E2 -10931.595} C_VEL
LIN {X 0,Y 404.124,Z 219.142,A -85,B 0,C 180,E1 -10934.519,E2 -10934.519} C_VEL
LIN {X 0,Y 404.177,Z 219.137,A -85,B 0,C 180,E1 -10937.3,E2 -10937.3} C_VEL
LIN {X 0,Y 404.14,Z 219.144,A -85,B 0,C 180,E1 -10939.951,E2 -10939.951} C_VEL
LIN {X 0,Y 404.107,Z 219.145,A -85,B 0,C 180,E1 -10943.121,E2 -10943.121} C_VEL
LIN {X 0,Y 404.11,Z 219.145,A -85,B 0,C 180,E1 -10946.184,E2 -10946.184} C_VEL
LIN {X 0,Y 404.115,Z 219.148,A -85,B 0,C 180,E1 -10949.712,E2 -10949.712} C_VEL
LIN {X 0,Y 404.156,Z 219.14,A -85,B 0,C 180,E1 -10953.12,E2 -10953.12} C_VEL
LIN {X 0,Y 404.139,Z 219.14,A -85,B 0,C 180,E1 -10956.423,E2 -10956.423} C_VEL
LIN {X 0,Y 404.183,Z 219.136,A -85,B 0,C 180,E1 -10959.858,E2 -10959.858} C_VEL
LIN {X 0,Y 404.173,Z 219.138,A -85,B 0,C 180,E1 -10962.99,E2 -10962.99} C_VEL
LIN {X 0,Y 404.221,Z 219.131,A -85,B 0,C 180,E1 -10966.787,E2 -10966.787} C_VEL
LIN {X 0,Y 404.227,Z 219.129,A -85,B 0,C 180,E1 -10969.987,E2 -10969.987} C_VEL
LIN {X 0,Y 404.395,Z 219.113,A -85,B 0,C 180,E1 -10973.012,E2 -10973.012} C_VEL
LIN {X 0,Y 404.241,Z 219.132,A -85,B 0,C 180,E1 -10975.013,E2 -10975.013} C_VEL
LIN {X 0,Y 404.431,Z 219.103,A -85,B 0,C 180,E1 -10978.008,E2 -10978.008} C_VEL
LIN {X 0,Y 404.56,Z 219.087,A -85,B 0,C 180,E1 -10980,E2 -10980} C_VEL
LIN {X 0,Y 404.365,Z 219.118,A -85,B 0,C 180,E1 -10982.989,E2 -10982.989} C_VEL
LIN {X 0,Y 404.341,Z 219.118,A -85,B 0,C 180,E1 -10986.71,E2 -10986.71} C_VEL
LIN {X 0,Y 404.243,Z 219.133,A -85,B 0,C 180,E1 -10989.002,E2 -10989.002} C_VEL
LIN {X 0,Y 404.221,Z 219.13,A -85,B 0,C 180,E1 -10992.042,E2 -10992.042} C_VEL
LIN {X 0,Y 404.161,Z 219.14,A -85,B 0,C 180,E1 -10995.119,E2 -10995.119} C_VEL
LIN {X 0,Y 404.163,Z 219.138,A -85,B 0,C 180,E1 -10998.24,E2 -10998.24} C_VEL
LIN {X 0,Y 404.092,Z 219.146,A -85,B 0,C 180,E1 -11001.422,E2 -11001.422} C_VEL
LIN {X 0,Y 404.131,Z 219.148,A -85,B 0,C 180,E1 -11004.668,E2 -11004.668} C_VEL
LIN {X 0,Y 404.154,Z 219.139,A -85,B 0,C 180,E1 -11008.002,E2 -11008.002} C_VEL
LIN {X 0,Y 404.099,Z 219.145,A -85,B 0,C 180,E1 -11011.56,E2 -11011.56} C_VEL
LIN {X 0,Y 404.147,Z 219.14,A -85,B 0,C 180,E1 -11015.019,E2 -11015.019} C_VEL
LIN {X 0,Y 404.114,Z 219.146,A -85,B 0,C 180,E1 -11018.761,E2 -11018.761} C_VEL
LIN {X 0,Y 404.089,Z 219.146,A -85,B 0,C 180,E1 -11021.603,E2 -11021.603} C_VEL
LIN {X 0,Y 404.115,Z 219.147,A -85,B 0,C 180,E1 -11024.525,E2 -11024.525} C_VEL
LIN {X 0,Y 404.108,Z 219.144,A -85,B 0,C 180,E1 -11027.299,E2 -11027.299} C_VEL
LIN {X 0,Y 404.144,Z 219.143,A -85,B 0,C 180,E1 -11029.959,E2 -11029.959} C_VEL
LIN {X 0,Y 404.114,Z 219.143,A -85,B 0,C 180,E1 -11033.129,E2 -11033.129} C_VEL
LIN {X 0,Y 404.125,Z 219.148,A -85,B 0,C 180,E1 -11036.191,E2 -11036.191} C_VEL
LIN {X 0,Y 404.128,Z 219.144,A -85,B 0,C 180,E1 -11039.719,E2 -11039.719} C_VEL
LIN {X 0,Y 404.18,Z 219.135,A -85,B 0,C 180,E1 -11043.126,E2 -11043.126} C_VEL
LIN {X 0,Y 404.16,Z 219.138,A -85,B 0,C 180,E1 -11045.338,E2 -11045.338} C_VEL
LIN {X 0,Y 404.127,Z 219.142,A -85,B 0,C 180,E1 -11048.584,E2 -11048.584} C_VEL
LIN {X 0,Y 404.195,Z 219.139,A -85,B 0,C 180,E1 -11051.765,E2 -11051.765} C_VEL
LIN {X 0,Y 404.197,Z 219.132,A -85,B 0,C 180,E1 -11054.885,E2 -11054.885} C_VEL
LIN {X 0,Y 404.25,Z 219.13,A -85,B 0,C 180,E1 -11057.961,E2 -11057.961} C_VEL
LIN {X 0,Y 404.261,Z 219.125,A -85,B 0,C 180,E1 -11061.001,E2 -11061.001} C_VEL
LIN {X 0,Y 404.389,Z 219.243,A -85,B 0,C 180,E1 -11063.579,E2 -11063.579} C_VEL
LIN {X 0,Y 405.878,Z 228.817,A -85,B 0,C 180,E1 -11065.797,E2 -11065.797} C_VEL
LIN {X 0,Y 409.844,Z 249.65,A -85,B 0,C 180,E1 -11066.338,E2 -11066.338} C_VEL
LIN {X 0,Y 408.663,Z 336.384,A -85,B 0,C 180,E1 -11067.885,E2 -11067.885} C_VEL
LIN {X 0,Y 408.3,Z 349.547,A -85,B 0,C 180,E1 -11068.323,E2 -11068.323} C_VEL
LIN {X 0,Y 407.847,Z 361.627,A -85,B 0,C 180,E1 -11068.915,E2 -11068.915} C_VEL
LIN {X 0,Y 407.259,Z 373.86,A -85,B 0,C 180,E1 -11069.73,E2 -11069.73} C_VEL
LIN {X 0,Y 407.152,Z 375.467,A -85,B 0,C 180,E1 -11069.856,E2 -11069.856} C_VEL
LIN {X 0,Y 406.158,Z 380.596,A -85,B 0,C 180,E1 -11070.257,E2 -11070.257} C_VEL
LIN {X 0,Y 402.771,Z 388.638,A -85,B 0,C 180,E1 -11070.935,E2 -11070.935} C_VEL
LIN {X 0,Y 399.428,Z 396.234,A -85,B 0,C 180,E1 -11071.704,E2 -11071.704} C_VEL
LIN {X 0,Y 398.481,Z 400.593,A -85,B 0,C 180,E1 -11072.25,E2 -11072.25} C_VEL
LIN {X 0,Y 397.755,Z 409.216,A -85,B 0,C 180,E1 -11073.547,E2 -11073.547} C_VEL
LIN {X 0,Y 397.18,Z 417.423,A -85,B 0,C 180,E1 -11075.077,E2 -11075.077} C_VEL
LIN {X 0,Y 396.785,Z 423.976,A -85,B 0,C 180,E1 -11076.598,E2 -11076.598} C_VEL
LIN {X 0,Y 396.385,Z 429.326,A -85,B 0,C 180,E1 -11078.155,E2 -11078.155} C_VEL
LIN {X 0,Y 396.089,Z 433.444,A -85,B 0,C 180,E1 -11079.705,E2 -11079.705} C_VEL
LIN {X 0,Y 395.937,Z 436.489,A -85,B 0,C 180,E1 -11081.26,E2 -11081.26} C_VEL
LIN {X 0,Y 395.84,Z 438.128,A -85,B 0,C 180,E1 -11082.446,E2 -11082.446} C_VEL
LIN {X 0,Y 395.721,Z 439.658,A -85,B 0,C 180,E1 -11084.397,E2 -11084.397} C_VEL
LIN {X 0,Y 395.737,Z 439.896,A -85,B 0,C 180,E1 -11085.45,E2 -11085.45} C_VEL
LIN {X 0,Y 395.74,Z 439.674,A -85,B 0,C 180,E1 -11086.508,E2 -11086.508} C_VEL
LIN {X 0,Y 395.782,Z 439.042,A -85,B 0,C 180,E1 -11087.57,E2 -11087.57} C_VEL
LIN {X 0,Y 395.899,Z 437.997,A -85,B 0,C 180,E1 -11088.635,E2 -11088.635} C_VEL
LIN {X 0,Y 396.136,Z 436.128,A -85,B 0,C 180,E1 -11089.9,E2 -11089.9} C_VEL
LIN {X 0,Y 396.497,Z 432.013,A -85,B 0,C 180,E1 -11091.853,E2 -11091.853} C_VEL
LIN {X 0,Y 396.978,Z 427.25,A -85,B 0,C 180,E1 -11093.474,E2 -11093.474} C_VEL
LIN {X 0,Y 397.627,Z 421.082,A -85,B 0,C 180,E1 -11095.099,E2 -11095.099} C_VEL
LIN {X 0,Y 398.406,Z 413.272,A -85,B 0,C 180,E1 -11096.732,E2 -11096.732} C_VEL
LIN {X 0,Y 399.262,Z 405.194,A -85,B 0,C 180,E1 -11098.09,E2 -11098.09} C_VEL
LIN {X 0,Y 400.187,Z 395.129,A -85,B 0,C 180,E1 -11099.453,E2 -11099.453} C_VEL
LIN {X 0,Y 401.277,Z 383.768,A -85,B 0,C 180,E1 -11100.675,E2 -11100.675} C_VEL
LIN {X 0,Y 402.164,Z 372.604,A -85,B 0,C 180,E1 -11101.617,E2 -11101.617} C_VEL
LIN {X 0,Y 402.936,Z 360.012,A -85,B 0,C 180,E1 -11102.434,E2 -11102.434} C_VEL
LIN {X 0,Y 403.527,Z 347.204,A -85,B 0,C 180,E1 -11103.036,E2 -11103.036} C_VEL
LIN {X 0,Y 403.885,Z 334.082,A -85,B 0,C 180,E1 -11103.43,E2 -11103.43} C_VEL
LIN {X 0,Y 405.261,Z 250.601,A -85,B 0,C 180,E1 -11104.949,E2 -11104.949} C_VEL
LIN {X 0,Y 401.95,Z 236.521,A -85,B 0,C 180,E1 -11105.428,E2 -11105.428} C_VEL
LIN {X 0,Y 399.122,Z 229.261,A -85,B 0,C 180,E1 -11105.782,E2 -11105.782} C_VEL
LIN {X 0,Y 397.136,Z 220.019,A -85,B 0,C 180,E1 -11108.141,E2 -11108.141} C_VEL
LIN {X 0,Y 397.145,Z 220.012,A -85,B 0,C 180,E1 -11111.992,E2 -11111.992} C_VEL
LIN {X 0,Y 397.139,Z 220.016,A -85,B 0,C 180,E1 -11115.058,E2 -11115.058} C_VEL
LIN {X 0,Y 397.143,Z 220.015,A -85,B 0,C 180,E1 -11118.006,E2 -11118.006} C_VEL
LIN {X 0,Y 397.093,Z 220.023,A -85,B 0,C 180,E1 -11121.724,E2 -11121.724} C_VEL
LIN {X 0,Y 397.108,Z 220.015,A -85,B 0,C 180,E1 -11125.505,E2 -11125.505} C_VEL
LIN {X 0,Y 397.064,Z 220.02,A -85,B 0,C 180,E1 -11129.117,E2 -11129.117} C_VEL
LIN {X 0,Y 397.175,Z 220.007,A -85,B 0,C 180,E1 -11132.609,E2 -11132.609} C_VEL
LIN {X 0,Y 397.114,Z 220.016,A -85,B 0,C 180,E1 -11135.981,E2 -11135.981} C_VEL
LIN {X 0,Y 397.136,Z 220.012,A -85,B 0,C 180,E1 -11139.697,E2 -11139.697} C_VEL
LIN {X 0,Y 397.161,Z 220.005,A -85,B 0,C 180,E1 -11142.844,E2 -11142.844} C_VEL
LIN {X 0,Y 397.204,Z 220.003,A -85,B 0,C 180,E1 -11146.679,E2 -11146.679} C_VEL
LIN {X 0,Y 397.192,Z 220.008,A -85,B 0,C 180,E1 -11149.809,E2 -11149.809} C_VEL
LIN {X 0,Y 397.333,Z 219.984,A -85,B 0,C 180,E1 -11152.888,E2 -11152.888} C_VEL
LIN {X 0,Y 397.229,Z 220.002,A -85,B 0,C 180,E1 -11154.925,E2 -11154.925} C_VEL
LIN {X 0,Y 397.42,Z 219.975,A -85,B 0,C 180,E1 -11157.973,E2 -11157.973} C_VEL
LIN {X 0,Y 397.551,Z 219.956,A -85,B 0,C 180,E1 -11160,E2 -11160} C_VEL
LIN {X 0,Y 397.346,Z 219.986,A -85,B 0,C 180,E1 -11163.042,E2 -11163.042} C_VEL
LIN {X 0,Y 397.304,Z 219.99,A -85,B 0,C 180,E1 -11167.113,E2 -11167.113} C_VEL
LIN {X 0,Y 397.197,Z 219.996,A -85,B 0,C 180,E1 -11170.192,E2 -11170.192} C_VEL
LIN {X 0,Y 397.205,Z 220.002,A -85,B 0,C 180,E1 -11173.322,E2 -11173.322} C_VEL
LIN {X 0,Y 397.164,Z 220.011,A -85,B 0,C 180,E1 -11177.158,E2 -11177.158} C_VEL
LIN {X 0,Y 397.077,Z 220.023,A -85,B 0,C 180,E1 -11180.732,E2 -11180.732} C_VEL
LIN {X 0,Y 397.094,Z 220.015,A -85,B 0,C 180,E1 -11184.021,E2 -11184.021} C_VEL
LIN {X 0,Y 397.067,Z 220.018,A -85,B 0,C 180,E1 -11187.756,E2 -11187.756} C_VEL
LIN {X 0,Y 397.058,Z 220.022,A -85,B 0,C 180,E1 -11190.885,E2 -11190.885} C_VEL
LIN {X 0,Y 397.101,Z 220.018,A -85,B 0,C 180,E1 -11194.496,E2 -11194.496} C_VEL
LIN {X 0,Y 397.082,Z 220.021,A -85,B 0,C 180,E1 -11198.278,E2 -11198.278} C_VEL
LIN {X 0,Y 397.05,Z 220.016,A -85,B 0,C 180,E1 -11200.914,E2 -11200.914} C_VEL
LIN {X 0,Y 397.09,Z 220.019,A -85,B 0,C 180,E1 -11203.651,E2 -11203.651} C_VEL
LIN {X 0,Y 397.092,Z 220.023,A -85,B 0,C 180,E1 -11206.523,E2 -11206.523} C_VEL
LIN {X 0,Y 397.08,Z 220.018,A -85,B 0,C 180,E1 -11210.421,E2 -11210.421} C_VEL
LIN {X 0,Y 397.091,Z 220.016,A -85,B 0,C 180,E1 -11213.006,E2 -11213.006} C_VEL
LIN {X 0,Y 397.116,Z 220.018,A -85,B 0,C 180,E1 -11216.283,E2 -11216.283} C_VEL
LIN {X 0,Y 397.111,Z 220.02,A -85,B 0,C 180,E1 -11220.17,E2 -11220.17} C_VEL
LIN {X 0,Y 399.598,Z 231.018,A -85,B 0,C 180,E1 -11222.789,E2 -11222.789} C_VEL
LIN {X 0,Y 401.13,Z 238.995,A -85,B 0,C 180,E1 -11224.58,E2 -11224.58} C_VEL
LIN {X 0,Y 400.932,Z 242.685,A -85,B 0,C 180,E1 -11225.336,E2 -11225.336} C_VEL
LIN {X 0,Y 399.679,Z 257.608,A -85,B 0,C 180,E1 -11228.33,E2 -11228.33} C_VEL
LIN {X 0,Y 399.333,Z 262.551,A -85,B 0,C 180,E1 -11229.314,E2 -11229.314} C_VEL
LIN {X 0,Y 403.429,Z 285.123,A -85,B 0,C 180,E1 -11230.008,E2 -11230.008} C_VEL
LIN {X 0,Y 404.683,Z 295.021,A -85,B 0,C 180,E1 -11230.271,E2 -11230.271} C_VEL
LIN {X 0,Y 403.469,Z 372.193,A -85,B 0,C 180,E1 -11231.697,E2 -11231.697} C_VEL
LIN {X 0,Y 402.82,Z 385.804,A -85,B 0,C 180,E1 -11232.157,E2 -11232.157} C_VEL
LIN {X 0,Y 401.995,Z 398.158,A -85,B 0,C 180,E1 -11232.775,E2 -11232.775} C_VEL
LIN {X 0,Y 400.973,Z 410.011,A -85,B 0,C 180,E1 -11233.583,E2 -11233.583} C_VEL
LIN {X 0,Y 399.978,Z 421.408,A -85,B 0,C 180,E1 -11234.587,E2 -11234.587} C_VEL
LIN {X 0,Y 398.994,Z 431.713,A -85,B 0,C 180,E1 -11235.723,E2 -11235.723} C_VEL
LIN {X 0,Y 398.197,Z 440.998,A -85,B 0,C 180,E1 -11236.995,E2 -11236.995} C_VEL
LIN {X 0,Y 397.25,Z 450.025,A -85,B 0,C 180,E1 -11238.519,E2 -11238.519} C_VEL
LIN {X 0,Y 396.624,Z 457.325,A -85,B 0,C 180,E1 -11240.05,E2 -11240.05} C_VEL
LIN {X 0,Y 396.161,Z 464.038,A -85,B 0,C 180,E1 -11241.84,E2 -11241.84} C_VEL
LIN {X 0,Y 395.877,Z 468.618,A -85,B 0,C 180,E1 -11243.424,E2 -11243.424} C_VEL
LIN {X 0,Y 395.83,Z 471.882,A -85,B 0,C 180,E1 -11244.906,E2 -11244.906} C_VEL
LIN {X 0,Y 395.765,Z 474.866,A -85,B 0,C 180,E1 -11246.945,E2 -11246.945} C_VEL
LIN {X 0,Y 395.857,Z 475.764,A -85,B 0,C 180,E1 -11247.964,E2 -11247.964} C_VEL
LIN {X 0,Y 395.833,Z 476.221,A -85,B 0,C 180,E1 -11248.981,E2 -11248.981} C_VEL
LIN {X 0,Y 395.823,Z 476.281,A -85,B 0,C 180,E1 -11249.998,E2 -11249.998} C_VEL
LIN {X 0,Y 395.877,Z 475.238,A -85,B 0,C 180,E1 -11252.033,E2 -11252.033} C_VEL
LIN {X 0,Y 395.789,Z 474.073,A -85,B 0,C 180,E1 -11253.052,E2 -11253.052} C_VEL
LIN {X 0,Y 395.828,Z 471.556,A -85,B 0,C 180,E1 -11254.581,E2 -11254.581} C_VEL
LIN {X 0,Y 395.929,Z 466.714,A -85,B 0,C 180,E1 -11256.572,E2 -11256.572} C_VEL
LIN {X 0,Y 396.109,Z 461.51,A -85,B 0,C 180,E1 -11258.158,E2 -11258.158} C_VEL
LIN {X 0,Y 396.436,Z 455.143,A -85,B 0,C 180,E1 -11259.693,E2 -11259.693} C_VEL
LIN {X 0,Y 396.962,Z 447.154,A -85,B 0,C 180,E1 -11261.227,E2 -11261.227} C_VEL
LIN {X 0,Y 397.566,Z 439.008,A -85,B 0,C 180,E1 -11262.504,E2 -11262.504} C_VEL
LIN {X 0,Y 398.327,Z 428.747,A -85,B 0,C 180,E1 -11263.815,E2 -11263.815} C_VEL
LIN {X 0,Y 399.057,Z 417.901,A -85,B 0,C 180,E1 -11264.923,E2 -11264.923} C_VEL
LIN {X 0,Y 399.85,Z 406.963,A -85,B 0,C 180,E1 -11265.806,E2 -11265.806} C_VEL
LIN {X 0,Y 400.556,Z 394.88,A -85,B 0,C 180,E1 -11266.562,E2 -11266.562} C_VEL
LIN {X 0,Y 401.179,Z 382.54,A -85,B 0,C 180,E1 -11267.126,E2 -11267.126} C_VEL
LIN {X 0,Y 401.662,Z 369.889,A -85,B 0,C 180,E1 -11267.498,E2 -11267.498} C_VEL
LIN {X 0,Y 402.391,Z 292.141,A -85,B 0,C 180,E1 -11268.906,E2 -11268.906} C_VEL
LIN {X 0,Y 398.419,Z 263.206,A -85,B 0,C 180,E1 -11269.612,E2 -11269.612} C_VEL
LIN {X 0,Y 399.632,Z 244.286,A -85,B 0,C 180,E1 -11273.305,E2 -11273.305} C_VEL
LIN {X 0,Y 400.118,Z 236.052,A -85,B 0,C 180,E1 -11274.928,E2 -11274.928} C_VEL
LIN {X 0,Y 398.455,Z 226.187,A -85,B 0,C 180,E1 -11277.007,E2 -11277.007} C_VEL
LIN {X 0,Y 397.181,Z 220.014,A -85,B 0,C 180,E1 -11278.344,E2 -11278.344} C_VEL
LIN {X 0,Y 397.064,Z 220.028,A -85,B 0,C 180,E1 -11282.068,E2 -11282.068} C_VEL
LIN {X 0,Y 397.102,Z 220.018,A -85,B 0,C 180,E1 -11285.499,E2 -11285.499} C_VEL
LIN {X 0,Y 397.109,Z 220.016,A -85,B 0,C 180,E1 -11288.857,E2 -11288.857} C_VEL
LIN {X 0,Y 397.044,Z 220.026,A -85,B 0,C 180,E1 -11292.263,E2 -11292.263} C_VEL
LIN {X 0,Y 397.084,Z 220.019,A -85,B 0,C 180,E1 -11295.061,E2 -11295.061} C_VEL
LIN {X 0,Y 397.127,Z 220.018,A -85,B 0,C 180,E1 -11298.003,E2 -11298.003} C_VEL
LIN {X 0,Y 397.079,Z 220.026,A -85,B 0,C 180,E1 -11301.722,E2 -11301.722} C_VEL
LIN {X 0,Y 397.091,Z 220.023,A -85,B 0,C 180,E1 -11305.503,E2 -11305.503} C_VEL
LIN {X 0,Y 397.046,Z 220.025,A -85,B 0,C 180,E1 -11309.114,E2 -11309.114} C_VEL
LIN {X 0,Y 397.156,Z 220.01,A -85,B 0,C 180,E1 -11312.607,E2 -11312.607} C_VEL
LIN {X 0,Y 397.098,Z 220.019,A -85,B 0,C 180,E1 -11315.979,E2 -11315.979} C_VEL
LIN {X 0,Y 397.112,Z 220.02,A -85,B 0,C 180,E1 -11319.27,E2 -11319.27} C_VEL
LIN {X 0,Y 397.139,Z 220.013,A -85,B 0,C 180,E1 -11322.842,E2 -11322.842} C_VEL
LIN {X 0,Y 397.137,Z 220.015,A -85,B 0,C 180,E1 -11325.655,E2 -11325.655} C_VEL
LIN {X 0,Y 397.164,Z 220.01,A -85,B 0,C 180,E1 -11328.775,E2 -11328.775} C_VEL
LIN {X 0,Y 397.352,Z 219.985,A -85,B 0,C 180,E1 -11332.036,E2 -11332.036} C_VEL
LIN {X 0,Y 397.349,Z 219.986,A -85,B 0,C 180,E1 -11333.908,E2 -11333.908} C_VEL
LIN {X 0,Y 397.4,Z 219.979,A -85,B 0,C 180,E1 -11337.973,E2 -11337.973} C_VEL
LIN {X 0,Y 397.53,Z 219.963,A -85,B 0,C 180,E1 -11340,E2 -11340} C_VEL
LIN {X 0,Y 397.325,Z 219.996,A -85,B 0,C 180,E1 -11343.042,E2 -11343.042} C_VEL
LIN {X 0,Y 397.292,Z 219.994,A -85,B 0,C 180,E1 -11346.709,E2 -11346.709} C_VEL
LIN {X 0,Y 397.205,Z 220.008,A -85,B 0,C 180,E1 -11349.163,E2 -11349.163} C_VEL
LIN {X 0,Y 397.181,Z 220.008,A -85,B 0,C 180,E1 -11352.259,E2 -11352.259} C_VEL
LIN {X 0,Y 397.135,Z 220.014,A -85,B 0,C 180,E1 -11355.393,E2 -11355.393} C_VEL
LIN {X 0,Y 397.115,Z 220.02,A -85,B 0,C 180,E1 -11358.575,E2 -11358.575} C_VEL
LIN {X 0,Y 397.05,Z 220.023,A -85,B 0,C 180,E1 -11361.821,E2 -11361.821} C_VEL
LIN {X 0,Y 397.11,Z 220.015,A -85,B 0,C 180,E1 -11365.514,E2 -11365.514} C_VEL
LIN {X 0,Y 397.075,Z 220.026,A -85,B 0,C 180,E1 -11368.547,E2 -11368.547} C_VEL
LIN {X 0,Y 397.038,Z 220.026,A -85,B 0,C 180,E1 -11372.075,E2 -11372.075} C_VEL
LIN {X 0,Y 397.083,Z 220.019,A -85,B 0,C 180,E1 -11375.506,E2 -11375.506} C_VEL
LIN {X 0,Y 397.09,Z 220.02,A -85,B 0,C 180,E1 -11378.864,E2 -11378.864} C_VEL
LIN {X 0,Y 397.036,Z 220.031,A -85,B 0,C 180,E1 -11382.271,E2 -11382.271} C_VEL
LIN {X 0,Y 397.057,Z 220.022,A -85,B 0,C 180,E1 -11385.073,E2 -11385.073} C_VEL
LIN {X 0,Y 397.039,Z 220.028,A -85,B 0,C 180,E1 -11388.025,E2 -11388.025} C_VEL
LIN {X 0,Y 397.107,Z 220.016,A -85,B 0,C 180,E1 -11391.142,E2 -11391.142} C_VEL
LIN {X 0,Y 397.098,Z 220.02,A -85,B 0,C 180,E1 -11394.501,E2 -11394.501} C_VEL
LIN {X 0,Y 397.06,Z 220.027,A -85,B 0,C 180,E1 -11397.932,E2 -11397.932} C_VEL
LIN {X 0,Y 397.105,Z 220.017,A -85,B 0,C 180,E1 -11401.46,E2 -11401.46} C_VEL
LIN {X 0,Y 397.138,Z 220.013,A -85,B 0,C 180,E1 -11404.491,E2 -11404.491} C_VEL
LIN {X 0,Y 397.084,Z 220.022,A -85,B 0,C 180,E1 -11408.185,E2 -11408.185} C_VEL
LIN {X 0,Y 397.148,Z 220.013,A -85,B 0,C 180,E1 -11411.43,E2 -11411.43} C_VEL
LIN {X 0,Y 397.17,Z 220.008,A -85,B 0,C 180,E1 -11414.611,E2 -11414.611} C_VEL
LIN {X 0,Y 397.213,Z 220.01,A -85,B 0,C 180,E1 -11417.745,E2 -11417.745} C_VEL
LIN {X 0,Y 397.231,Z 220,A -85,B 0,C 180,E1 -11420.84,E2 -11420.84} C_VEL
LIN {X 0,Y 397.373,Z 220.195,A -85,B 0,C 180,E1 -11423.401,E2 -11423.401} C_VEL
LIN {X 0,Y 398.833,Z 229.063,A -85,B 0,C 180,E1 -11425.501,E2 -11425.501} C_VEL
LIN {X 0,Y 403.022,Z 249.727,A -85,B 0,C 180,E1 -11426.061,E2 -11426.061} C_VEL
LIN {X 0,Y 401.807,Z 336.143,A -85,B 0,C 180,E1 -11427.621,E2 -11427.621} C_VEL
LIN {X 0,Y 401.44,Z 349.727,A -85,B 0,C 180,E1 -11428.076,E2 -11428.076} C_VEL
LIN {X 0,Y 400.933,Z 362.54,A -85,B 0,C 180,E1 -11428.716,E2 -11428.716} C_VEL
LIN {X 0,Y 400.397,Z 373.391,A -85,B 0,C 180,E1 -11429.449,E2 -11429.449} C_VEL
LIN {X 0,Y 399.637,Z 384.251,A -85,B 0,C 180,E1 -11430.38,E2 -11430.38} C_VEL
LIN {X 0,Y 398.901,Z 394.819,A -85,B 0,C 180,E1 -11431.516,E2 -11431.516} C_VEL
LIN {X 0,Y 398.481,Z 400.593,A -85,B 0,C 180,E1 -11432.25,E2 -11432.25} C_VEL
LIN {X 0,Y 397.56,Z 404.849,A -85,B 0,C 180,E1 -11432.824,E2 -11432.824} C_VEL
LIN {X 0,Y 394.263,Z 411.357,A -85,B 0,C 180,E1 -11433.796,E2 -11433.796} C_VEL
LIN {X 0,Y 390.902,Z 417.243,A -85,B 0,C 180,E1 -11434.858,E2 -11434.858} C_VEL
LIN {X 0,Y 389.9,Z 420.53,A -85,B 0,C 180,E1 -11435.566,E2 -11435.566} C_VEL
LIN {X 0,Y 389.498,Z 427.02,A -85,B 0,C 180,E1 -11437.257,E2 -11437.257} C_VEL
LIN {X 0,Y 389.161,Z 431.737,A -85,B 0,C 180,E1 -11438.831,E2 -11438.831} C_VEL
LIN {X 0,Y 388.893,Z 435.341,A -85,B 0,C 180,E1 -11440.412,E2 -11440.412} C_VEL
LIN {X 0,Y 388.82,Z 437.166,A -85,B 0,C 180,E1 -11441.469,E2 -11441.469} C_VEL
LIN {X 0,Y 388.736,Z 438.541,A -85,B 0,C 180,E1 -11442.531,E2 -11442.531} C_VEL
LIN {X 0,Y 388.665,Z 439.517,A -85,B 0,C 180,E1 -11443.596,E2 -11443.596} C_VEL
LIN {X 0,Y 388.623,Z 440.087,A -85,B 0,C 180,E1 -11444.666,E2 -11444.666} C_VEL
LIN {X 0,Y 388.65,Z 440.006,A -85,B 0,C 180,E1 -11446.584,E2 -11446.584} C_VEL
LIN {X 0,Y 388.739,Z 439.2,A -85,B 0,C 180,E1 -11447.899,E2 -11447.899} C_VEL
LIN {X 0,Y 388.895,Z 438.038,A -85,B 0,C 180,E1 -11448.983,E2 -11448.983} C_VEL
LIN {X 0,Y 389.179,Z 435.444,A -85,B 0,C 180,E1 -11450.618,E2 -11450.618} C_VEL
LIN {X 0,Y 389.535,Z 431.735,A -85,B 0,C 180,E1 -11452.264,E2 -11452.264} C_VEL
LIN {X 0,Y 390.072,Z 426.784,A -85,B 0,C 180,E1 -11453.915,E2 -11453.915} C_VEL
LIN {X 0,Y 390.778,Z 420.424,A -85,B 0,C 180,E1 -11455.571,E2 -11455.571} C_VEL
LIN {X 0,Y 391.509,Z 413.83,A -85,B 0,C 180,E1 -11456.953,E2 -11456.953} C_VEL
LIN {X 0,Y 392.362,Z 406.076,A -85,B 0,C 180,E1 -11458.29,E2 -11458.29} C_VEL
LIN {X 0,Y 393.303,Z 396.958,A -85,B 0,C 180,E1 -11459.579,E2 -11459.579} C_VEL
LIN {X 0,Y 394.357,Z 385.951,A -85,B 0,C 180,E1 -11460.82,E2 -11460.82} C_VEL
LIN {X 0,Y 395.367,Z 374.854,A -85,B 0,C 180,E1 -11461.812,E2 -11461.812} C_VEL
LIN {X 0,Y 396.13,Z 363.539,A -85,B 0,C 180,E1 -11462.608,E2 -11462.608} C_VEL
LIN {X 0,Y 396.799,Z 350.431,A -85,B 0,C 180,E1 -11463.282,E2 -11463.282} C_VEL
LIN {X 0,Y 397.238,Z 337.052,A -85,B 0,C 180,E1 -11463.744,E2 -11463.744} C_VEL
LIN {X 0,Y 398.711,Z 251.442,A -85,B 0,C 180,E1 -11465.344,E2 -11465.344} C_VEL
LIN {X 0,Y 395.771,Z 239.083,A -85,B 0,C 180,E1 -11465.777,E2 -11465.777} C_VEL
LIN {X 0,Y 392.018,Z 229.717,A -85,B 0,C 180,E1 -11466.221,E2 -11466.221} C_VEL
LIN {X 0,Y 390.071,Z 220.899,A -85,B 0,C 180,E1 -11468.513,E2 -11468.513} C_VEL
LIN {X 0,Y 390.094,Z 220.889,A -85,B 0,C 180,E1 -11471.803,E2 -11471.803} C_VEL
LIN {X 0,Y 390.107,Z 220.892,A -85,B 0,C 180,E1 -11475.364,E2 -11475.364} C_VEL
LIN {X 0,Y 390.091,Z 220.894,A -85,B 0,C 180,E1 -11478.195,E2 -11478.195} C_VEL
LIN {X 0,Y 390.08,Z 220.894,A -85,B 0,C 180,E1 -11480.907,E2 -11480.907} C_VEL
LIN {X 0,Y 390.069,Z 220.891,A -85,B 0,C 180,E1 -11484.792,E2 -11484.792} C_VEL
LIN {X 0,Y 390.008,Z 220.9,A -85,B 0,C 180,E1 -11488.495,E2 -11488.495} C_VEL
LIN {X 0,Y 390.099,Z 220.888,A -85,B 0,C 180,E1 -11492.069,E2 -11492.069} C_VEL
LIN {X 0,Y 390.06,Z 220.89,A -85,B 0,C 180,E1 -11495.518,E2 -11495.518} C_VEL
LIN {X 0,Y 390.061,Z 220.888,A -85,B 0,C 180,E1 -11498.878,E2 -11498.878} C_VEL
LIN {X 0,Y 390.109,Z 220.885,A -85,B 0,C 180,E1 -11502.166,E2 -11502.166} C_VEL
LIN {X 0,Y 390.122,Z 220.891,A -85,B 0,C 180,E1 -11505.392,E2 -11505.392} C_VEL
LIN {X 0,Y 390.121,Z 220.885,A -85,B 0,C 180,E1 -11508.571,E2 -11508.571} C_VEL
LIN {X 0,Y 390.285,Z 220.861,A -85,B 0,C 180,E1 -11512.031,E2 -11512.031} C_VEL
LIN {X 0,Y 390.201,Z 220.877,A -85,B 0,C 180,E1 -11514.833,E2 -11514.833} C_VEL
LIN {X 0,Y 390.39,Z 220.851,A -85,B 0,C 180,E1 -11517.937,E2 -11517.937} C_VEL
LIN {X 0,Y 390.521,Z 220.831,A -85,B 0,C 180,E1 -11520,E2 -11520} C_VEL
LIN {X 0,Y 390.28,Z 220.867,A -85,B 0,C 180,E1 -11523.097,E2 -11523.097} C_VEL
LIN {X 0,Y 390.276,Z 220.858,A -85,B 0,C 180,E1 -11526.203,E2 -11526.203} C_VEL
LIN {X 0,Y 390.17,Z 220.875,A -85,B 0,C 180,E1 -11529.33,E2 -11529.33} C_VEL
LIN {X 0,Y 390.154,Z 220.881,A -85,B 0,C 180,E1 -11532.484,E2 -11532.484} C_VEL
LIN {X 0,Y 390.117,Z 220.884,A -85,B 0,C 180,E1 -11535.678,E2 -11535.678} C_VEL
LIN {X 0,Y 390.074,Z 220.89,A -85,B 0,C 180,E1 -11538.924,E2 -11538.924} C_VEL
LIN {X 0,Y 390.014,Z 220.901,A -85,B 0,C 180,E1 -11542.236,E2 -11542.236} C_VEL
LIN {X 0,Y 390.032,Z 220.898,A -85,B 0,C 180,E1 -11545.724,E2 -11545.724} C_VEL
LIN {X 0,Y 390.012,Z 220.903,A -85,B 0,C 180,E1 -11549.114,E2 -11549.114} C_VEL
LIN {X 0,Y 390.024,Z 220.904,A -85,B 0,C 180,E1 -11552.724,E2 -11552.724} C_VEL
LIN {X 0,Y 390.028,Z 220.9,A -85,B 0,C 180,E1 -11555.824,E2 -11555.824} C_VEL
LIN {X 0,Y 390.03,Z 220.9,A -85,B 0,C 180,E1 -11559.215,E2 -11559.215} C_VEL
LIN {X 0,Y 390.027,Z 220.89,A -85,B 0,C 180,E1 -11562.375,E2 -11562.375} C_VEL
LIN {X 0,Y 390.034,Z 220.898,A -85,B 0,C 180,E1 -11565.356,E2 -11565.356} C_VEL
LIN {X 0,Y 390.012,Z 220.905,A -85,B 0,C 180,E1 -11568.187,E2 -11568.187} C_VEL
LIN {X 0,Y 390.052,Z 220.897,A -85,B 0,C 180,E1 -11570.905,E2 -11570.905} C_VEL
LIN {X 0,Y 390.081,Z 220.896,A -85,B 0,C 180,E1 -11574.794,E2 -11574.794} C_VEL
LIN {X 0,Y 390.021,Z 220.903,A -85,B 0,C 180,E1 -11578.497,E2 -11578.497} C_VEL
LIN {X 0,Y 390.056,Z 220.905,A -85,B 0,C 180,E1 -11579.802,E2 -11579.802} C_VEL
LIN {X 0,Y 392.678,Z 232.366,A -85,B 0,C 180,E1 -11582.558,E2 -11582.558} C_VEL
LIN {X 0,Y 394.232,Z 240.316,A -85,B 0,C 180,E1 -11584.387,E2 -11584.387} C_VEL
LIN {X 0,Y 394.181,Z 242.86,A -85,B 0,C 180,E1 -11584.925,E2 -11584.925} C_VEL
LIN {X 0,Y 392.774,Z 258.594,A -85,B 0,C 180,E1 -11588.138,E2 -11588.138} C_VEL
LIN {X 0,Y 392.499,Z 262.312,A -85,B 0,C 180,E1 -11588.878,E2 -11588.878} C_VEL
LIN {X 0,Y 396.608,Z 284.421,A -85,B 0,C 180,E1 -11589.577,E2 -11589.577} C_VEL
LIN {X 0,Y 398.129,Z 295.395,A -85,B 0,C 180,E1 -11589.886,E2 -11589.886} C_VEL
LIN {X 0,Y 396.873,Z 371.65,A -85,B 0,C 180,E1 -11591.318,E2 -11591.318} C_VEL
LIN {X 0,Y 396.299,Z 384.494,A -85,B 0,C 180,E1 -11591.753,E2 -11591.753} C_VEL
LIN {X 0,Y 395.404,Z 396.56,A -85,B 0,C 180,E1 -11592.346,E2 -11592.346} C_VEL
LIN {X 0,Y 394.347,Z 408.778,A -85,B 0,C 180,E1 -11593.165,E2 -11593.165} C_VEL
LIN {X 0,Y 393.271,Z 420.34,A -85,B 0,C 180,E1 -11594.185,E2 -11594.185} C_VEL
LIN {X 0,Y 392.241,Z 430.974,A -85,B 0,C 180,E1 -11595.365,E2 -11595.365} C_VEL
LIN {X 0,Y 391.417,Z 439.32,A -85,B 0,C 180,E1 -11596.501,E2 -11596.501} C_VEL
LIN {X 0,Y 390.624,Z 447.227,A -85,B 0,C 180,E1 -11597.795,E2 -11597.795} C_VEL
LIN {X 0,Y 389.806,Z 454.987,A -85,B 0,C 180,E1 -11599.35,E2 -11599.35} C_VEL
LIN {X 0,Y 389.226,Z 462.145,A -85,B 0,C 180,E1 -11601.17,E2 -11601.17} C_VEL
LIN {X 0,Y 388.905,Z 466.939,A -85,B 0,C 180,E1 -11602.732,E2 -11602.732} C_VEL
LIN {X 0,Y 388.753,Z 469.786,A -85,B 0,C 180,E1 -11603.887,E2 -11603.887} C_VEL
LIN {X 0,Y 388.7,Z 473.315,A -85,B 0,C 180,E1 -11605.851,E2 -11605.851} C_VEL
LIN {X 0,Y 388.754,Z 475.465,A -85,B 0,C 180,E1 -11607.926,E2 -11607.926} C_VEL
LIN {X 0,Y 388.762,Z 475.901,A -85,B 0,C 180,E1 -11608.962,E2 -11608.962} C_VEL
LIN {X 0,Y 388.751,Z 475.946,A -85,B 0,C 180,E1 -11609.998,E2 -11609.998} C_VEL
LIN {X 0,Y 388.762,Z 475.604,A -85,B 0,C 180,E1 -11611.034,E2 -11611.034} C_VEL
LIN {X 0,Y 388.79,Z 474.868,A -85,B 0,C 180,E1 -11612.07,E2 -11612.07} C_VEL
LIN {X 0,Y 388.692,Z 473.675,A -85,B 0,C 180,E1 -11613.107,E2 -11613.107} C_VEL
LIN {X 0,Y 388.762,Z 471.128,A -85,B 0,C 180,E1 -11614.664,E2 -11614.664} C_VEL
LIN {X 0,Y 388.794,Z 467.546,A -85,B 0,C 180,E1 -11616.224,E2 -11616.224} C_VEL
LIN {X 0,Y 388.966,Z 462.84,A -85,B 0,C 180,E1 -11617.786,E2 -11617.786} C_VEL
LIN {X 0,Y 389.271,Z 456.863,A -85,B 0,C 180,E1 -11619.349,E2 -11619.349} C_VEL
LIN {X 0,Y 389.727,Z 449.397,A -85,B 0,C 180,E1 -11620.912,E2 -11620.912} C_VEL
LIN {X 0,Y 390.442,Z 440.114,A -85,B 0,C 180,E1 -11622.471,E2 -11622.471} C_VEL
LIN {X 0,Y 391.195,Z 430.82,A -85,B 0,C 180,E1 -11623.723,E2 -11623.723} C_VEL
LIN {X 0,Y 391.97,Z 419.713,A -85,B 0,C 180,E1 -11624.933,E2 -11624.933} C_VEL
LIN {X 0,Y 392.69,Z 409.34,A -85,B 0,C 180,E1 -11625.835,E2 -11625.835} C_VEL
LIN {X 0,Y 393.507,Z 396.97,A -85,B 0,C 180,E1 -11626.668,E2 -11626.668} C_VEL
LIN {X 0,Y 394.241,Z 383.952,A -85,B 0,C 180,E1 -11627.303,E2 -11627.303} C_VEL
LIN {X 0,Y 394.76,Z 371.334,A -85,B 0,C 180,E1 -11627.714,E2 -11627.714} C_VEL
LIN {X 0,Y 395.609,Z 293.229,A -85,B 0,C 180,E1 -11629.158,E2 -11629.158} C_VEL
LIN {X 0,Y 391.487,Z 262.888,A -85,B 0,C 180,E1 -11629.91,E2 -11629.91} C_VEL
LIN {X 0,Y 392.757,Z 243.733,A -85,B 0,C 180,E1 -11633.717,E2 -11633.717} C_VEL
LIN {X 0,Y 393.105,Z 236.756,A -85,B 0,C 180,E1 -11635.121,E2 -11635.121} C_VEL
LIN {X 0,Y 391.101,Z 225.459,A -85,B 0,C 180,E1 -11637.558,E2 -11637.558} C_VEL
LIN {X 0,Y 390.14,Z 220.891,A -85,B 0,C 180,E1 -11638.621,E2 -11638.621} C_VEL
LIN {X 0,Y 390.028,Z 220.898,A -85,B 0,C 180,E1 -11642.717,E2 -11642.717} C_VEL
LIN {X 0,Y 390.038,Z 220.901,A -85,B 0,C 180,E1 -11645.821,E2 -11645.821} C_VEL
LIN {X 0,Y 390.048,Z 220.896,A -85,B 0,C 180,E1 -11649.214,E2 -11649.214} C_VEL
LIN {X 0,Y 390.018,Z 220.901,A -85,B 0,C 180,E1 -11652.37,E2 -11652.37} C_VEL
LIN {X 0,Y 390.072,Z 220.896,A -85,B 0,C 180,E1 -11656.103,E2 -11656.103} C_VEL
LIN {X 0,Y 390.054,Z 220.895,A -85,B 0,C 180,E1 -11659.17,E2 -11659.17} C_VEL
LIN {X 0,Y 390.015,Z 220.9,A -85,B 0,C 180,E1 -11662.445,E2 -11662.445} C_VEL
LIN {X 0,Y 390.033,Z 220.9,A -85,B 0,C 180,E1 -11666.041,E2 -11666.041} C_VEL
LIN {X 0,Y 390.014,Z 220.903,A -85,B 0,C 180,E1 -11669.865,E2 -11669.865} C_VEL
LIN {X 0,Y 390.074,Z 220.895,A -85,B 0,C 180,E1 -11673.229,E2 -11673.229} C_VEL
LIN {X 0,Y 390.079,Z 220.892,A -85,B 0,C 180,E1 -11676.743,E2 -11676.743} C_VEL
LIN {X 0,Y 390.087,Z 220.892,A -85,B 0,C 180,E1 -11679.982,E2 -11679.982} C_VEL
LIN {X 0,Y 390.096,Z 220.895,A -85,B 0,C 180,E1 -11683.246,E2 -11683.246} C_VEL
LIN {X 0,Y 390.15,Z 220.883,A -85,B 0,C 180,E1 -11686.56,E2 -11686.56} C_VEL
LIN {X 0,Y 390.133,Z 220.887,A -85,B 0,C 180,E1 -11689.622,E2 -11689.622} C_VEL
LIN {X 0,Y 390.294,Z 220.867,A -85,B 0,C 180,E1 -11692.758,E2 -11692.758} C_VEL
LIN {X 0,Y 390.186,Z 220.881,A -85,B 0,C 180,E1 -11694.833,E2 -11694.833} C_VEL
LIN {X 0,Y 390.369,Z 220.855,A -85,B 0,C 180,E1 -11697.936,E2 -11697.936} C_VEL
LIN {X 0,Y 390.5,Z 220.839,A -85,B 0,C 180,E1 -11700,E2 -11700} C_VEL
LIN {X 0,Y 390.26,Z 220.875,A -85,B 0,C 180,E1 -11703.097,E2 -11703.097} C_VEL
LIN {X 0,Y 390.246,Z 220.87,A -85,B 0,C 180,E1 -11706.705,E2 -11706.705} C_VEL
LIN {X 0,Y 390.158,Z 220.884,A -85,B 0,C 180,E1 -11709.33,E2 -11709.33} C_VEL
LIN {X 0,Y 390.13,Z 220.888,A -85,B 0,C 180,E1 -11712.484,E2 -11712.484} C_VEL
LIN {X 0,Y 390.095,Z 220.889,A -85,B 0,C 180,E1 -11715.678,E2 -11715.678} C_VEL
LIN {X 0,Y 390.054,Z 220.899,A -85,B 0,C 180,E1 -11718.924,E2 -11718.924} C_VEL
LIN {X 0,Y 389.992,Z 220.904,A -85,B 0,C 180,E1 -11722.237,E2 -11722.237} C_VEL
LIN {X 0,Y 390.077,Z 220.892,A -85,B 0,C 180,E1 -11725.745,E2 -11725.745} C_VEL
LIN {X 0,Y 390.012,Z 220.901,A -85,B 0,C 180,E1 -11729.113,E2 -11729.113} C_VEL
LIN {X 0,Y 390.004,Z 220.905,A -85,B 0,C 180,E1 -11732.725,E2 -11732.725} C_VEL
LIN {X 0,Y 390.019,Z 220.9,A -85,B 0,C 180,E1 -11735.828,E2 -11735.828} C_VEL
LIN {X 0,Y 390.027,Z 220.898,A -85,B 0,C 180,E1 -11739.22,E2 -11739.22} C_VEL
LIN {X 0,Y 390.01,Z 220.907,A -85,B 0,C 180,E1 -11742.377,E2 -11742.377} C_VEL
LIN {X 0,Y 390.015,Z 220.899,A -85,B 0,C 180,E1 -11745.358,E2 -11745.358} C_VEL
LIN {X 0,Y 390.004,Z 220.907,A -85,B 0,C 180,E1 -11748.19,E2 -11748.19} C_VEL
LIN {X 0,Y 390.067,Z 220.893,A -85,B 0,C 180,E1 -11750.911,E2 -11750.911} C_VEL
LIN {X 0,Y 390.064,Z 220.894,A -85,B 0,C 180,E1 -11754.797,E2 -11754.797} C_VEL
LIN {X 0,Y 390.005,Z 220.903,A -85,B 0,C 180,E1 -11758.499,E2 -11758.499} C_VEL
LIN {X 0,Y 390.102,Z 220.895,A -85,B 0,C 180,E1 -11762.074,E2 -11762.074} C_VEL
LIN {X 0,Y 390.064,Z 220.895,A -85,B 0,C 180,E1 -11765.523,E2 -11765.523} C_VEL
LIN {X 0,Y 390.077,Z 220.894,A -85,B 0,C 180,E1 -11769.533,E2 -11769.533} C_VEL
LIN {X 0,Y 390.13,Z 220.886,A -85,B 0,C 180,E1 -11773.251,E2 -11773.251} C_VEL
LIN {X 0,Y 390.188,Z 220.878,A -85,B 0,C 180,E1 -11776.564,E2 -11776.564} C_VEL
LIN {X 0,Y 390.162,Z 220.887,A -85,B 0,C 180,E1 -11779.625,E2 -11779.625} C_VEL
LIN {X 0,Y 390.332,Z 220.997,A -85,B 0,C 180,E1 -11783.184,E2 -11783.184} C_VEL
LIN {X 0,Y 391.711,Z 229.222,A -85,B 0,C 180,E1 -11785.178,E2 -11785.178} C_VEL
LIN {X 0,Y 394.736,Z 243.188,A -85,B 0,C 180,E1 -11785.588,E2 -11785.588} C_VEL
LIN {X 0,Y 396.19,Z 250.789,A -85,B 0,C 180,E1 -11785.793,E2 -11785.793} C_VEL
LIN {X 0,Y 394.931,Z 337.227,A -85,B 0,C 180,E1 -11787.388,E2 -11787.388} C_VEL
LIN {X 0,Y 394.548,Z 350.876,A -85,B 0,C 180,E1 -11787.865,E2 -11787.865} C_VEL
LIN {X 0,Y 394.044,Z 362.929,A -85,B 0,C 180,E1 -11788.485,E2 -11788.485} C_VEL
LIN {X 0,Y 393.421,Z 374.782,A -85,B 0,C 180,E1 -11789.312,E2 -11789.312} C_VEL
LIN {X 0,Y 392.56,Z 386.718,A -85,B 0,C 180,E1 -11790.386,E2 -11790.386} C_VEL
LIN {X 0,Y 391.788,Z 396.91,A -85,B 0,C 180,E1 -11791.544,E2 -11791.544} C_VEL
LIN {X 0,Y 391.072,Z 406.068,A -85,B 0,C 180,E1 -11792.834,E2 -11792.834} C_VEL
LIN {X 0,Y 390.36,Z 414.993,A -85,B 0,C 180,E1 -11794.39,E2 -11794.39} C_VEL
LIN {X 0,Y 389.9,Z 420.53,A -85,B 0,C 180,E1 -11795.566,E2 -11795.566} C_VEL
LIN {X 0,Y 388.94,Z 423.622,A -85,B 0,C 180,E1 -11796.297,E2 -11796.297} C_VEL
LIN {X 0,Y 385.773,Z 428.221,A -85,B 0,C 180,E1 -11797.511,E2 -11797.511} C_VEL
LIN {X 0,Y 382.709,Z 432.118,A -85,B 0,C 180,E1 -11798.795,E2 -11798.795} C_VEL
LIN {X 0,Y 381.926,Z 434.086,A -85,B 0,C 180,E1 -11799.623,E2 -11799.623} C_VEL
LIN {X 0,Y 381.79,Z 436.09,A -85,B 0,C 180,E1 -11800.608,E2 -11800.608} C_VEL
LIN {X 0,Y 381.637,Z 438.905,A -85,B 0,C 180,E1 -11802.575,E2 -11802.575} C_VEL
LIN {X 0,Y 381.557,Z 440.014,A -85,B 0,C 180,E1 -11803.855,E2 -11803.855} C_VEL
LIN {X 0,Y 381.523,Z 440.459,A -85,B 0,C 180,E1 -11804.946,E2 -11804.946} C_VEL
LIN {X 0,Y 381.567,Z 440.318,A -85,B 0,C 180,E1 -11806.71,E2 -11806.71} C_VEL
LIN {X 0,Y 381.695,Z 439.322,A -85,B 0,C 180,E1 -11808.241,E2 -11808.241} C_VEL
LIN {X 0,Y 382.047,Z 436.693,A -85,B 0,C 180,E1 -11810.253,E2 -11810.253} C_VEL
LIN {X 0,Y 382.427,Z 432.881,A -85,B 0,C 180,E1 -11812.131,E2 -11812.131} C_VEL
LIN {X 0,Y 382.971,Z 428.2,A -85,B 0,C 180,E1 -11813.811,E2 -11813.811} C_VEL
LIN {X 0,Y 383.713,Z 422.114,A -85,B 0,C 180,E1 -11815.494,E2 -11815.494} C_VEL
LIN {X 0,Y 384.615,Z 414.396,A -85,B 0,C 180,E1 -11817.181,E2 -11817.181} C_VEL
LIN {X 0,Y 385.648,Z 405.628,A -85,B 0,C 180,E1 -11818.714,E2 -11818.714} C_VEL
LIN {X 0,Y 386.685,Z 395.413,A -85,B 0,C 180,E1 -11820.137,E2 -11820.137} C_VEL
LIN {X 0,Y 387.744,Z 385.407,A -85,B 0,C 180,E1 -11821.253,E2 -11821.253} C_VEL
LIN {X 0,Y 388.713,Z 375.203,A -85,B 0,C 180,E1 -11822.171,E2 -11822.171} C_VEL
LIN {X 0,Y 389.546,Z 363.569,A -85,B 0,C 180,E1 -11822.998,E2 -11822.998} C_VEL
LIN {X 0,Y 390.241,Z 350.756,A -85,B 0,C 180,E1 -11823.665,E2 -11823.665} C_VEL
LIN {X 0,Y 390.66,Z 338.023,A -85,B 0,C 180,E1 -11824.116,E2 -11824.116} C_VEL
LIN {X 0,Y 392.222,Z 252.61,A -85,B 0,C 180,E1 -11825.743,E2 -11825.743} C_VEL
LIN {X 0,Y 389.497,Z 241.249,A -85,B 0,C 180,E1 -11826.155,E2 -11826.155} C_VEL
LIN {X 0,Y 384.883,Z 230.018,A -85,B 0,C 180,E1 -11826.726,E2 -11826.726} C_VEL
LIN {X 0,Y 383.056,Z 221.774,A -85,B 0,C 180,E1 -11828.93,E2 -11828.93} C_VEL
LIN {X 0,Y 383.056,Z 221.775,A -85,B 0,C 180,E1 -11832.787,E2 -11832.787} C_VEL
LIN {X 0,Y 383.06,Z 221.77,A -85,B 0,C 180,E1 -11835.799,E2 -11835.799} C_VEL
LIN {X 0,Y 383.031,Z 221.773,A -85,B 0,C 180,E1 -11838.785,E2 -11838.785} C_VEL
LIN {X 0,Y 382.988,Z 221.777,A -85,B 0,C 180,E1 -11842.095,E2 -11842.095} C_VEL
LIN {X 0,Y 383.002,Z 221.771,A -85,B 0,C 180,E1 -11845.331,E2 -11845.331} C_VEL
LIN {X 0,Y 382.967,Z 221.776,A -85,B 0,C 180,E1 -11849.08,E2 -11849.08} C_VEL
LIN {X 0,Y 383.038,Z 221.768,A -85,B 0,C 180,E1 -11852.697,E2 -11852.697} C_VEL
LIN {X 0,Y 383.023,Z 221.772,A -85,B 0,C 180,E1 -11856.192,E2 -11856.192} C_VEL
LIN {X 0,Y 383.051,Z 221.764,A -85,B 0,C 180,E1 -11859.599,E2 -11859.599} C_VEL
LIN {X 0,Y 383.084,Z 221.759,A -85,B 0,C 180,E1 -11862.931,E2 -11862.931} C_VEL
LIN {X 0,Y 383.103,Z 221.759,A -85,B 0,C 180,E1 -11866.464,E2 -11866.464} C_VEL
LIN {X 0,Y 383.127,Z 221.757,A -85,B 0,C 180,E1 -11870.498,E2 -11870.498} C_VEL
LIN {X 0,Y 383.235,Z 221.738,A -85,B 0,C 180,E1 -11872.625,E2 -11872.625} C_VEL
LIN {X 0,Y 383.174,Z 221.752,A -85,B 0,C 180,E1 -11874.738,E2 -11874.738} C_VEL
LIN {X 0,Y 383.358,Z 221.727,A -85,B 0,C 180,E1 -11877.899,E2 -11877.899} C_VEL
LIN {X 0,Y 383.491,Z 221.707,A -85,B 0,C 180,E1 -11880,E2 -11880} C_VEL
LIN {X 0,Y 383.217,Z 221.747,A -85,B 0,C 180,E1 -11883.154,E2 -11883.154} C_VEL
LIN {X 0,Y 383.234,Z 221.735,A -85,B 0,C 180,E1 -11886.317,E2 -11886.317} C_VEL
LIN {X 0,Y 383.121,Z 221.751,A -85,B 0,C 180,E1 -11889.503,E2 -11889.503} C_VEL
LIN {X 0,Y 383.119,Z 221.76,A -85,B 0,C 180,E1 -11892.717,E2 -11892.717} C_VEL
LIN {X 0,Y 383.059,Z 221.763,A -85,B 0,C 180,E1 -11895.975,E2 -11895.975} C_VEL
LIN {X 0,Y 383.027,Z 221.767,A -85,B 0,C 180,E1 -11899.286,E2 -11899.286} C_VEL
LIN {X 0,Y 382.969,Z 221.777,A -85,B 0,C 180,E1 -11902.668,E2 -11902.668} C_VEL
LIN {X 0,Y 382.972,Z 221.78,A -85,B 0,C 180,E1 -11906.132,E2 -11906.132} C_VEL
LIN {X 0,Y 382.96,Z 221.78,A -85,B 0,C 180,E1 -11909.703,E2 -11909.703} C_VEL
LIN {X 0,Y 382.984,Z 221.776,A -85,B 0,C 180,E1 -11913.403,E2 -11913.403} C_VEL
LIN {X 0,Y 383.008,Z 221.777,A -85,B 0,C 180,E1 -11916.164,E2 -11916.164} C_VEL
LIN {X 0,Y 382.976,Z 221.781,A -85,B 0,C 180,E1 -11919.963,E2 -11919.963} C_VEL
LIN {X 0,Y 382.997,Z 221.77,A -85,B 0,C 180,E1 -11922.78,E2 -11922.78} C_VEL
LIN {X 0,Y 382.987,Z 221.777,A -85,B 0,C 180,E1 -11925.79,E2 -11925.79} C_VEL
LIN {X 0,Y 382.956,Z 221.781,A -85,B 0,C 180,E1 -11928.802,E2 -11928.802} C_VEL
LIN {X 0,Y 382.988,Z 221.78,A -85,B 0,C 180,E1 -11932.099,E2 -11932.099} C_VEL
LIN {X 0,Y 383.015,Z 221.774,A -85,B 0,C 180,E1 -11935.333,E2 -11935.333} C_VEL
LIN {X 0,Y 382.98,Z 221.781,A -85,B 0,C 180,E1 -11939.082,E2 -11939.082} C_VEL
LIN {X 0,Y 382.997,Z 221.823,A -85,B 0,C 180,E1 -11939.389,E2 -11939.389} C_VEL
LIN {X 0,Y 385.515,Z 232.391,A -85,B 0,C 180,E1 -11942.004,E2 -11942.004} C_VEL
LIN {X 0,Y 387.324,Z 241.662,A -85,B 0,C 180,E1 -11944.185,E2 -11944.185} C_VEL
LIN {X 0,Y 387.318,Z 244.316,A -85,B 0,C 180,E1 -11944.761,E2 -11944.761} C_VEL
LIN {X 0,Y 385.984,Z 258.756,A -85,B 0,C 180,E1 -11947.769,E2 -11947.769} C_VEL
LIN {X 0,Y 385.715,Z 261.786,A -85,B 0,C 180,E1 -11948.394,E2 -11948.394} C_VEL
LIN {X 0,Y 389.869,Z 283.722,A -85,B 0,C 180,E1 -11949.132,E2 -11949.132} C_VEL
LIN {X 0,Y 391.594,Z 296.609,A -85,B 0,C 180,E1 -11949.499,E2 -11949.499} C_VEL
LIN {X 0,Y 390.3,Z 371.177,A -85,B 0,C 180,E1 -11950.923,E2 -11950.923} C_VEL
LIN {X 0,Y 389.702,Z 384.068,A -85,B 0,C 180,E1 -11951.364,E2 -11951.364} C_VEL
LIN {X 0,Y 388.767,Z 396.146,A -85,B 0,C 180,E1 -11951.966,E2 -11951.966} C_VEL
LIN {X 0,Y 387.769,Z 407.555,A -85,B 0,C 180,E1 -11952.735,E2 -11952.735} C_VEL
LIN {X 0,Y 386.594,Z 419.295,A -85,B 0,C 180,E1 -11953.769,E2 -11953.769} C_VEL
LIN {X 0,Y 385.502,Z 429.836,A -85,B 0,C 180,E1 -11954.942,E2 -11954.942} C_VEL
LIN {X 0,Y 384.505,Z 439.369,A -85,B 0,C 180,E1 -11956.254,E2 -11956.254} C_VEL
LIN {X 0,Y 383.499,Z 448.584,A -85,B 0,C 180,E1 -11957.833,E2 -11957.833} C_VEL
LIN {X 0,Y 382.684,Z 456.017,A -85,B 0,C 180,E1 -11959.417,E2 -11959.417} C_VEL
LIN {X 0,Y 382.185,Z 462.008,A -85,B 0,C 180,E1 -11961.006,E2 -11961.006} C_VEL
LIN {X 0,Y 381.84,Z 466.761,A -85,B 0,C 180,E1 -11962.596,E2 -11962.596} C_VEL
LIN {X 0,Y 381.666,Z 469.856,A -85,B 0,C 180,E1 -11963.913,E2 -11963.913} C_VEL
LIN {X 0,Y 381.624,Z 473.064,A -85,B 0,C 180,E1 -11965.774,E2 -11965.774} C_VEL
LIN {X 0,Y 381.577,Z 474.321,A -85,B 0,C 180,E1 -11966.831,E2 -11966.831} C_VEL
LIN {X 0,Y 381.653,Z 475.164,A -85,B 0,C 180,E1 -11967.888,E2 -11967.888} C_VEL
LIN {X 0,Y 381.693,Z 475.582,A -85,B 0,C 180,E1 -11968.943,E2 -11968.943} C_VEL
LIN {X 0,Y 381.694,Z 475.252,A -85,B 0,C 180,E1 -11971.053,E2 -11971.053} C_VEL
LIN {X 0,Y 381.689,Z 474.487,A -85,B 0,C 180,E1 -11972.108,E2 -11972.108} C_VEL
LIN {X 0,Y 381.644,Z 471.652,A -85,B 0,C 180,E1 -11974.222,E2 -11974.222} C_VEL
LIN {X 0,Y 381.69,Z 467.64,A -85,B 0,C 180,E1 -11976.121,E2 -11976.121} C_VEL
LIN {X 0,Y 381.885,Z 462.312,A -85,B 0,C 180,E1 -11977.931,E2 -11977.931} C_VEL
LIN {X 0,Y 382.275,Z 455.155,A -85,B 0,C 180,E1 -11979.788,E2 -11979.788} C_VEL
LIN {X 0,Y 382.829,Z 447.371,A -85,B 0,C 180,E1 -11981.379,E2 -11981.379} C_VEL
LIN {X 0,Y 383.433,Z 439.389,A -85,B 0,C 180,E1 -11982.703,E2 -11982.703} C_VEL
LIN {X 0,Y 384.268,Z 429.3,A -85,B 0,C 180,E1 -11984.064,E2 -11984.064} C_VEL
LIN {X 0,Y 385.035,Z 418.809,A -85,B 0,C 180,E1 -11985.208,E2 -11985.208} C_VEL
LIN {X 0,Y 385.848,Z 408.301,A -85,B 0,C 180,E1 -11986.124,E2 -11986.124} C_VEL
LIN {X 0,Y 386.592,Z 396.777,A -85,B 0,C 180,E1 -11986.907,E2 -11986.907} C_VEL
LIN {X 0,Y 387.346,Z 383.805,A -85,B 0,C 180,E1 -11987.553,E2 -11987.553} C_VEL
LIN {X 0,Y 387.889,Z 371.289,A -85,B 0,C 180,E1 -11987.97,E2 -11987.97} C_VEL
LIN {X 0,Y 388.82,Z 294.243,A -85,B 0,C 180,E1 -11989.42,E2 -11989.42} C_VEL
LIN {X 0,Y 384.517,Z 262.603,A -85,B 0,C 180,E1 -11990.213,E2 -11990.213} C_VEL
LIN {X 0,Y 385.86,Z 243.682,A -85,B 0,C 180,E1 -11994.041,E2 -11994.041} C_VEL
LIN {X 0,Y 386.089,Z 237.461,A -85,B 0,C 180,E1 -11995.322,E2 -11995.322} C_VEL
LIN {X 0,Y 384.007,Z 226.144,A -85,B 0,C 180,E1 -11997.815,E2 -11997.815} C_VEL
LIN {X 0,Y 383.067,Z 221.772,A -85,B 0,C 180,E1 -11998.822,E2 -11998.822} C_VEL
LIN {X 0,Y 382.972,Z 221.779,A -85,B 0,C 180,E1 -12002.418,E2 -12002.418} C_VEL
LIN {X 0,Y 383.007,Z 221.779,A -85,B 0,C 180,E1 -12005.951,E2 -12005.951} C_VEL
LIN {X 0,Y 382.994,Z 221.777,A -85,B 0,C 180,E1 -12009.582,E2 -12009.582} C_VEL
LIN {X 0,Y 382.983,Z 221.775,A -85,B 0,C 180,E1 -12012.774,E2 -12012.774} C_VEL
LIN {X 0,Y 383.008,Z 221.779,A -85,B 0,C 180,E1 -12015.79,E2 -12015.79} C_VEL
LIN {X 0,Y 383.016,Z 221.771,A -85,B 0,C 180,E1 -12018.782,E2 -12018.782} C_VEL
LIN {X 0,Y 382.972,Z 221.779,A -85,B 0,C 180,E1 -12022.092,E2 -12022.092} C_VEL
LIN {X 0,Y 382.985,Z 221.778,A -85,B 0,C 180,E1 -12025.328,E2 -12025.328} C_VEL
LIN {X 0,Y 382.949,Z 221.781,A -85,B 0,C 180,E1 -12029.078,E2 -12029.078} C_VEL
LIN {X 0,Y 383.019,Z 221.771,A -85,B 0,C 180,E1 -12032.695,E2 -12032.695} C_VEL
LIN {X 0,Y 383.007,Z 221.773,A -85,B 0,C 180,E1 -12036.191,E2 -12036.191} C_VEL
LIN {X 0,Y 383.039,Z 221.773,A -85,B 0,C 180,E1 -12039.597,E2 -12039.597} C_VEL
LIN {X 0,Y 383.062,Z 221.768,A -85,B 0,C 180,E1 -12042.929,E2 -12042.929} C_VEL
LIN {X 0,Y 383.081,Z 221.763,A -85,B 0,C 180,E1 -12046.462,E2 -12046.462} C_VEL
LIN {X 0,Y 383.096,Z 221.766,A -85,B 0,C 180,E1 -12049.429,E2 -12049.429} C_VEL
LIN {X 0,Y 383.245,Z 221.744,A -85,B 0,C 180,E1 -12052.624,E2 -12052.624} C_VEL
LIN {X 0,Y 383.159,Z 221.756,A -85,B 0,C 180,E1 -12054.738,E2 -12054.738} C_VEL
LIN {X 0,Y 383.337,Z 221.731,A -85,B 0,C 180,E1 -12057.898,E2 -12057.898} C_VEL
LIN {X 0,Y 383.47,Z 221.715,A -85,B 0,C 180,E1 -12060,E2 -12060} C_VEL
LIN {X 0,Y 383.196,Z 221.754,A -85,B 0,C 180,E1 -12063.154,E2 -12063.154} C_VEL
LIN {X 0,Y 383.205,Z 221.747,A -85,B 0,C 180,E1 -12066.699,E2 -12066.699} C_VEL
LIN {X 0,Y 383.105,Z 221.761,A -85,B 0,C 180,E1 -12069.503,E2 -12069.503} C_VEL
LIN {X 0,Y 383.094,Z 221.767,A -85,B 0,C 180,E1 -12072.717,E2 -12072.717} C_VEL
LIN {X 0,Y 383.036,Z 221.769,A -85,B 0,C 180,E1 -12075.975,E2 -12075.975} C_VEL
LIN {X 0,Y 383.006,Z 221.774,A -85,B 0,C 180,E1 -12079.286,E2 -12079.286} C_VEL
LIN {X 0,Y 382.948,Z 221.786,A -85,B 0,C 180,E1 -12082.668,E2 -12082.668} C_VEL
LIN {X 0,Y 383.039,Z 221.77,A -85,B 0,C 180,E1 -12086.126,E2 -12086.126} C_VEL
LIN {X 0,Y 382.948,Z 221.78,A -85,B 0,C 180,E1 -12089.703,E2 -12089.703} C_VEL
LIN {X 0,Y 382.965,Z 221.777,A -85,B 0,C 180,E1 -12093.404,E2 -12093.404} C_VEL
LIN {X 0,Y 382.996,Z 221.777,A -85,B 0,C 180,E1 -12096.167,E2 -12096.167} C_VEL
LIN {X 0,Y 382.973,Z 221.779,A -85,B 0,C 180,E1 -12099.962,E2 -12099.962} C_VEL
LIN {X 0,Y 382.976,Z 221.778,A -85,B 0,C 180,E1 -12102.782,E2 -12102.782} C_VEL
LIN {X 0,Y 382.968,Z 221.779,A -85,B 0,C 180,E1 -12105.793,E2 -12105.793} C_VEL
LIN {X 0,Y 382.962,Z 221.779,A -85,B 0,C 180,E1 -12108.8,E2 -12108.8} C_VEL
LIN {X 0,Y 382.977,Z 221.782,A -85,B 0,C 180,E1 -12112.1,E2 -12112.1} C_VEL
LIN {X 0,Y 382.998,Z 221.774,A -85,B 0,C 180,E1 -12115.336,E2 -12115.336} C_VEL
LIN {X 0,Y 382.965,Z 221.777,A -85,B 0,C 180,E1 -12119.085,E2 -12119.085} C_VEL
LIN {X 0,Y 383.042,Z 221.768,A -85,B 0,C 180,E1 -12122.702,E2 -12122.702} C_VEL
LIN {X 0,Y 383.037,Z 221.768,A -85,B 0,C 180,E1 -12125.043,E2 -12125.043} C_VEL
LIN {X 0,Y 382.981,Z 221.777,A -85,B 0,C 180,E1 -12128.472,E2 -12128.472} C_VEL
LIN {X 0,Y 383.043,Z 221.774,A -85,B 0,C 180,E1 -12131.829,E2 -12131.829} C_VEL
LIN {X 0,Y 383.102,Z 221.761,A -85,B 0,C 180,E1 -12135.121,E2 -12135.121} C_VEL
LIN {X 0,Y 383.091,Z 221.763,A -85,B 0,C 180,E1 -12138.361,E2 -12138.361} C_VEL
LIN {X 0,Y 383.216,Z 221.753,A -85,B 0,C 180,E1 -12142.025,E2 -12142.025} C_VEL
LIN {X 0,Y 383.29,Z 221.817,A -85,B 0,C 180,E1 -12142.959,E2 -12142.959} C_VEL
LIN {X 0,Y 384.628,Z 229.671,A -85,B 0,C 180,E1 -12144.879,E2 -12144.879} C_VEL
LIN {X 0,Y 386.841,Z 238.543,A -85,B 0,C 180,E1 -12145.15,E2 -12145.15} C_VEL
LIN {X 0,Y 389.369,Z 252.405,A -85,B 0,C 180,E1 -12145.527,E2 -12145.527} C_VEL
LIN {X 0,Y 388.094,Z 337.179,A -85,B 0,C 180,E1 -12147.115,E2 -12147.115} C_VEL
LIN {X 0,Y 387.705,Z 350.206,A -85,B 0,C 180,E1 -12147.567,E2 -12147.567} C_VEL
LIN {X 0,Y 387.166,Z 362.953,A -85,B 0,C 180,E1 -12148.223,E2 -12148.223} C_VEL
LIN {X 0,Y 386.517,Z 375.192,A -85,B 0,C 180,E1 -12149.09,E2 -12149.09} C_VEL
LIN {X 0,Y 385.674,Z 386.606,A -85,B 0,C 180,E1 -12150.132,E2 -12150.132} C_VEL
LIN {X 0,Y 384.862,Z 396.891,A -85,B 0,C 180,E1 -12151.31,E2 -12151.31} C_VEL
LIN {X 0,Y 384.118,Z 406.118,A -85,B 0,C 180,E1 -12152.623,E2 -12152.623} C_VEL
LIN {X 0,Y 383.343,Z 415.095,A -85,B 0,C 180,E1 -12154.207,E2 -12154.207} C_VEL
LIN {X 0,Y 382.738,Z 422.33,A -85,B 0,C 180,E1 -12155.798,E2 -12155.798} C_VEL
LIN {X 0,Y 382.374,Z 428.088,A -85,B 0,C 180,E1 -12157.393,E2 -12157.393} C_VEL
LIN {X 0,Y 382.057,Z 432.631,A -85,B 0,C 180,E1 -12158.997,E2 -12158.997} C_VEL
LIN {X 0,Y 381.926,Z 434.086,A -85,B 0,C 180,E1 -12159.623,E2 -12159.623} C_VEL
LIN {X 0,Y 381.148,Z 435.865,A -85,B 0,C 180,E1 -12160.465,E2 -12160.465} C_VEL
LIN {X 0,Y 378.152,Z 438.273,A -85,B 0,C 180,E1 -12161.846,E2 -12161.846} C_VEL
LIN {X 0,Y 375.651,Z 439.688,A -85,B 0,C 180,E1 -12162.978,E2 -12162.978} C_VEL
LIN {X 0,Y 374.552,Z 440.344,A -85,B 0,C 180,E1 -12163.864,E2 -12163.864} C_VEL
LIN {X 0,Y 374.447,Z 440.471,A -85,B 0,C 180,E1 -12164.166,E2 -12164.166} C_VEL
LIN {X 0,Y 374.429,Z 440.826,A -85,B 0,C 180,E1 -12165.235,E2 -12165.235} C_VEL
LIN {X 0,Y 374.499,Z 440.627,A -85,B 0,C 180,E1 -12166.847,E2 -12166.847} C_VEL
LIN {X 0,Y 374.666,Z 439.413,A -85,B 0,C 180,E1 -12168.596,E2 -12168.596} C_VEL
LIN {X 0,Y 374.993,Z 436.99,A -85,B 0,C 180,E1 -12170.434,E2 -12170.434} C_VEL
LIN {X 0,Y 375.344,Z 433.967,A -85,B 0,C 180,E1 -12171.992,E2 -12171.992} C_VEL
LIN {X 0,Y 375.933,Z 429.122,A -85,B 0,C 180,E1 -12173.84,E2 -12173.84} C_VEL
LIN {X 0,Y 376.607,Z 423.758,A -85,B 0,C 180,E1 -12175.417,E2 -12175.417} C_VEL
LIN {X 0,Y 377.541,Z 416.413,A -85,B 0,C 180,E1 -12177.133,E2 -12177.133} C_VEL
LIN {X 0,Y 378.48,Z 408.781,A -85,B 0,C 180,E1 -12178.564,E2 -12178.564} C_VEL
LIN {X 0,Y 379.552,Z 399.403,A -85,B 0,C 180,E1 -12179.996,E2 -12179.996} C_VEL
LIN {X 0,Y 380.714,Z 389.1,A -85,B 0,C 180,E1 -12181.261,E2 -12181.261} C_VEL
LIN {X 0,Y 381.772,Z 378.834,A -85,B 0,C 180,E1 -12182.265,E2 -12182.265} C_VEL
LIN {X 0,Y 382.722,Z 366.832,A -85,B 0,C 180,E1 -12183.191,E2 -12183.191} C_VEL
LIN {X 0,Y 383.499,Z 354.564,A -85,B 0,C 180,E1 -12183.902,E2 -12183.902} C_VEL
LIN {X 0,Y 384.032,Z 342.245,A -85,B 0,C 180,E1 -12184.403,E2 -12184.403} C_VEL
LIN {X 0,Y 384.324,Z 328.012,A -85,B 0,C 180,E1 -12184.749,E2 -12184.749} C_VEL
LIN {X 0,Y 385.822,Z 253.889,A -85,B 0,C 180,E1 -12186.152,E2 -12186.152} C_VEL
LIN {X 0,Y 383.288,Z 243.655,A -85,B 0,C 180,E1 -12186.54,E2 -12186.54} C_VEL
LIN {X 0,Y 377.739,Z 230.418,A -85,B 0,C 180,E1 -12187.229,E2 -12187.229} C_VEL
LIN {X 0,Y 375.988,Z 222.653,A -85,B 0,C 180,E1 -12189.379,E2 -12189.379} C_VEL
LIN {X 0,Y 375.986,Z 222.65,A -85,B 0,C 180,E1 -12192.29,E2 -12192.29} C_VEL
LIN {X 0,Y 376.005,Z 222.649,A -85,B 0,C 180,E1 -12195.254,E2 -12195.254} C_VEL
LIN {X 0,Y 375.987,Z 222.65,A -85,B 0,C 180,E1 -12199.14,E2 -12199.14} C_VEL
LIN {X 0,Y 375.953,Z 222.654,A -85,B 0,C 180,E1 -12201.911,E2 -12201.911} C_VEL
LIN {X 0,Y 375.964,Z 222.647,A -85,B 0,C 180,E1 -12205.332,E2 -12205.332} C_VEL
LIN {X 0,Y 375.941,Z 222.651,A -85,B 0,C 180,E1 -12208.437,E2 -12208.437} C_VEL
LIN {X 0,Y 375.978,Z 222.647,A -85,B 0,C 180,E1 -12212.14,E2 -12212.14} C_VEL
LIN {X 0,Y 375.986,Z 222.642,A -85,B 0,C 180,E1 -12214.538,E2 -12214.538} C_VEL
LIN {X 0,Y 375.96,Z 222.647,A -85,B 0,C 180,E1 -12218.046,E2 -12218.046} C_VEL
LIN {X 0,Y 376.008,Z 222.649,A -85,B 0,C 180,E1 -12221.474,E2 -12221.474} C_VEL
LIN {X 0,Y 376.037,Z 222.642,A -85,B 0,C 180,E1 -12224.832,E2 -12224.832} C_VEL
LIN {X 0,Y 376.024,Z 222.642,A -85,B 0,C 180,E1 -12228.136,E2 -12228.136} C_VEL
LIN {X 0,Y 376.198,Z 222.615,A -85,B 0,C 180,E1 -12231.918,E2 -12231.918} C_VEL
LIN {X 0,Y 376.146,Z 222.627,A -85,B 0,C 180,E1 -12234.64,E2 -12234.64} C_VEL
LIN {X 0,Y 376.324,Z 222.603,A -85,B 0,C 180,E1 -12237.86,E2 -12237.86} C_VEL
LIN {X 0,Y 376.461,Z 222.582,A -85,B 0,C 180,E1 -12240,E2 -12240} C_VEL
LIN {X 0,Y 376.155,Z 222.627,A -85,B 0,C 180,E1 -12243.214,E2 -12243.214} C_VEL
LIN {X 0,Y 376.193,Z 222.612,A -85,B 0,C 180,E1 -12246.436,E2 -12246.436} C_VEL
LIN {X 0,Y 376.092,Z 222.625,A -85,B 0,C 180,E1 -12249.682,E2 -12249.682} C_VEL
LIN {X 0,Y 376.069,Z 222.632,A -85,B 0,C 180,E1 -12253.658,E2 -12253.658} C_VEL
LIN {X 0,Y 376.013,Z 222.643,A -85,B 0,C 180,E1 -12257.401,E2 -12257.401} C_VEL
LIN {X 0,Y 375.961,Z 222.654,A -85,B 0,C 180,E1 -12260.833,E2 -12260.833} C_VEL
LIN {X 0,Y 375.951,Z 222.65,A -85,B 0,C 180,E1 -12264.285,E2 -12264.285} C_VEL
LIN {X 0,Y 375.912,Z 222.653,A -85,B 0,C 180,E1 -12267.866,E2 -12267.866} C_VEL
LIN {X 0,Y 375.921,Z 222.655,A -85,B 0,C 180,E1 -12270.69,E2 -12270.69} C_VEL
LIN {X 0,Y 375.943,Z 222.654,A -85,B 0,C 180,E1 -12274.114,E2 -12274.114} C_VEL
LIN {X 0,Y 375.936,Z 222.655,A -85,B 0,C 180,E1 -12276.744,E2 -12276.744} C_VEL
LIN {X 0,Y 375.958,Z 222.655,A -85,B 0,C 180,E1 -12279.968,E2 -12279.968} C_VEL
LIN {X 0,Y 375.92,Z 222.657,A -85,B 0,C 180,E1 -12283.768,E2 -12283.768} C_VEL
LIN {X 0,Y 375.927,Z 222.657,A -85,B 0,C 180,E1 -12286.812,E2 -12286.812} C_VEL
LIN {X 0,Y 375.929,Z 222.653,A -85,B 0,C 180,E1 -12290.535,E2 -12290.535} C_VEL
LIN {X 0,Y 375.959,Z 222.648,A -85,B 0,C 180,E1 -12293.497,E2 -12293.497} C_VEL
LIN {X 0,Y 375.957,Z 222.652,A -85,B 0,C 180,E1 -12295.89,E2 -12295.89} C_VEL
LIN {X 0,Y 375.972,Z 222.79,A -85,B 0,C 180,E1 -12298.966,E2 -12298.966} C_VEL
LIN {X 0,Y 378.601,Z 233.752,A -85,B 0,C 180,E1 -12301.748,E2 -12301.748} C_VEL
LIN {X 0,Y 380.42,Z 243.008,A -85,B 0,C 180,E1 -12303.975,E2 -12303.975} C_VEL
LIN {X 0,Y 380.468,Z 245.659,A -85,B 0,C 180,E1 -12304.566,E2 -12304.566} C_VEL
LIN {X 0,Y 379.056,Z 260.241,A -85,B 0,C 180,E1 -12307.661,E2 -12307.661} C_VEL
LIN {X 0,Y 378.924,Z 261.436,A -85,B 0,C 180,E1 -12307.911,E2 -12307.911} C_VEL
LIN {X 0,Y 383.09,Z 282.939,A -85,B 0,C 180,E1 -12308.663,E2 -12308.663} C_VEL
LIN {X 0,Y 385.081,Z 296.735,A -85,B 0,C 180,E1 -12309.078,E2 -12309.078} C_VEL
LIN {X 0,Y 383.749,Z 370.577,A -85,B 0,C 180,E1 -12310.509,E2 -12310.509} C_VEL
LIN {X 0,Y 383.131,Z 383.673,A -85,B 0,C 180,E1 -12310.963,E2 -12310.963} C_VEL
LIN {X 0,Y 382.167,Z 395.767,A -85,B 0,C 180,E1 -12311.574,E2 -12311.574} C_VEL
LIN {X 0,Y 381.025,Z 408.009,A -85,B 0,C 180,E1 -12312.42,E2 -12312.42} C_VEL
LIN {X 0,Y 379.79,Z 419.58,A -85,B 0,C 180,E1 -12313.47,E2 -12313.47} C_VEL
LIN {X 0,Y 378.656,Z 430.015,A -85,B 0,C 180,E1 -12314.663,E2 -12314.663} C_VEL
LIN {X 0,Y 377.603,Z 439.449,A -85,B 0,C 180,E1 -12315.997,E2 -12315.997} C_VEL
LIN {X 0,Y 376.547,Z 448.565,A -85,B 0,C 180,E1 -12317.605,E2 -12317.605} C_VEL
LIN {X 0,Y 375.666,Z 455.936,A -85,B 0,C 180,E1 -12319.217,E2 -12319.217} C_VEL
LIN {X 0,Y 375.143,Z 461.874,A -85,B 0,C 180,E1 -12320.836,E2 -12320.836} C_VEL
LIN {X 0,Y 374.758,Z 466.583,A -85,B 0,C 180,E1 -12322.456,E2 -12322.456} C_VEL
LIN {X 0,Y 374.58,Z 469.924,A -85,B 0,C 180,E1 -12323.939,E2 -12323.939} C_VEL
LIN {X 0,Y 374.549,Z 472.813,A -85,B 0,C 180,E1 -12325.694,E2 -12325.694} C_VEL
LIN {X 0,Y 374.489,Z 474.052,A -85,B 0,C 180,E1 -12326.771,E2 -12326.771} C_VEL
LIN {X 0,Y 374.552,Z 474.861,A -85,B 0,C 180,E1 -12327.848,E2 -12327.848} C_VEL
LIN {X 0,Y 374.624,Z 475.264,A -85,B 0,C 180,E1 -12328.923,E2 -12328.923} C_VEL
LIN {X 0,Y 374.611,Z 475.275,A -85,B 0,C 180,E1 -12329.998,E2 -12329.998} C_VEL
LIN {X 0,Y 374.626,Z 474.9,A -85,B 0,C 180,E1 -12331.073,E2 -12331.073} C_VEL
LIN {X 0,Y 374.589,Z 474.098,A -85,B 0,C 180,E1 -12332.148,E2 -12332.148} C_VEL
LIN {X 0,Y 374.575,Z 471.227,A -85,B 0,C 180,E1 -12334.302,E2 -12334.302} C_VEL
LIN {X 0,Y 374.592,Z 467.548,A -85,B 0,C 180,E1 -12336.078,E2 -12336.078} C_VEL
LIN {X 0,Y 374.753,Z 463.514,A -85,B 0,C 180,E1 -12337.541,E2 -12337.541} C_VEL
LIN {X 0,Y 375.015,Z 457.897,A -85,B 0,C 180,E1 -12339.163,E2 -12339.163} C_VEL
LIN {X 0,Y 375.457,Z 450.873,A -85,B 0,C 180,E1 -12340.786,E2 -12340.786} C_VEL
LIN {X 0,Y 376.24,Z 442.065,A -85,B 0,C 180,E1 -12342.402,E2 -12342.402} C_VEL
LIN {X 0,Y 377.072,Z 432.039,A -85,B 0,C 180,E1 -12343.881,E2 -12343.881} C_VEL
LIN {X 0,Y 377.842,Z 421.825,A -85,B 0,C 180,E1 -12345.091,E2 -12345.091} C_VEL
LIN {X 0,Y 378.697,Z 410.466,A -85,B 0,C 180,E1 -12346.16,E2 -12346.16} C_VEL
LIN {X 0,Y 379.546,Z 398.702,A -85,B 0,C 180,E1 -12347.022,E2 -12347.022} C_VEL
LIN {X 0,Y 380.356,Z 385.919,A -85,B 0,C 180,E1 -12347.712,E2 -12347.712} C_VEL
LIN {X 0,Y 380.914,Z 373.436,A -85,B 0,C 180,E1 -12348.172,E2 -12348.172} C_VEL
LIN {X 0,Y 381.296,Z 353.441,A -85,B 0,C 180,E1 -12348.594,E2 -12348.594} C_VEL
LIN {X 0,Y 381.922,Z 294.479,A -85,B 0,C 180,E1 -12349.709,E2 -12349.709} C_VEL
LIN {X 0,Y 377.577,Z 262.242,A -85,B 0,C 180,E1 -12350.539,E2 -12350.539} C_VEL
LIN {X 0,Y 378.982,Z 243.53,A -85,B 0,C 180,E1 -12354.398,E2 -12354.398} C_VEL
LIN {X 0,Y 379.046,Z 238.155,A -85,B 0,C 180,E1 -12355.532,E2 -12355.532} C_VEL
LIN {X 0,Y 376.721,Z 225.917,A -85,B 0,C 180,E1 -12358.289,E2 -12358.289} C_VEL
LIN {X 0,Y 376.003,Z 222.652,A -85,B 0,C 180,E1 -12359.071,E2 -12359.071} C_VEL
LIN {X 0,Y 375.934,Z 222.654,A -85,B 0,C 180,E1 -12362.824,E2 -12362.824} C_VEL
LIN {X 0,Y 375.94,Z 222.654,A -85,B 0,C 180,E1 -12365.411,E2 -12365.411} C_VEL
LIN {X 0,Y 375.954,Z 222.654,A -85,B 0,C 180,E1 -12368.266,E2 -12368.266} C_VEL
LIN {X 0,Y 375.911,Z 222.659,A -85,B 0,C 180,E1 -12371.596,E2 -12371.596} C_VEL
LIN {X 0,Y 375.95,Z 222.653,A -85,B 0,C 180,E1 -12375.257,E2 -12375.257} C_VEL
LIN {X 0,Y 375.962,Z 222.651,A -85,B 0,C 180,E1 -12378.386,E2 -12378.386} C_VEL
LIN {X 0,Y 375.937,Z 222.658,A -85,B 0,C 180,E1 -12381.908,E2 -12381.908} C_VEL
LIN {X 0,Y 375.947,Z 222.655,A -85,B 0,C 180,E1 -12385.329,E2 -12385.329} C_VEL
LIN {X 0,Y 375.923,Z 222.655,A -85,B 0,C 180,E1 -12388.434,E2 -12388.434} C_VEL
LIN {X 0,Y 375.959,Z 222.651,A -85,B 0,C 180,E1 -12392.138,E2 -12392.138} C_VEL
LIN {X 0,Y 375.968,Z 222.649,A -85,B 0,C 180,E1 -12394.536,E2 -12394.536} C_VEL
LIN {X 0,Y 375.963,Z 222.651,A -85,B 0,C 180,E1 -12398.045,E2 -12398.045} C_VEL
LIN {X 0,Y 375.988,Z 222.652,A -85,B 0,C 180,E1 -12401.472,E2 -12401.472} C_VEL
LIN {X 0,Y 376.017,Z 222.645,A -85,B 0,C 180,E1 -12404.831,E2 -12404.831} C_VEL
LIN {X 0,Y 376.013,Z 222.644,A -85,B 0,C 180,E1 -12408.135,E2 -12408.135} C_VEL
LIN {X 0,Y 376.219,Z 222.619,A -85,B 0,C 180,E1 -12411.87,E2 -12411.87} C_VEL
LIN {X 0,Y 376.132,Z 222.63,A -85,B 0,C 180,E1 -12414.639,E2 -12414.639} C_VEL
LIN {X 0,Y 376.304,Z 222.608,A -85,B 0,C 180,E1 -12417.859,E2 -12417.859} C_VEL
LIN {X 0,Y 376.44,Z 222.59,A -85,B 0,C 180,E1 -12420,E2 -12420} C_VEL
LIN {X 0,Y 376.135,Z 222.633,A -85,B 0,C 180,E1 -12423.213,E2 -12423.213} C_VEL
LIN {X 0,Y 376.169,Z 222.624,A -85,B 0,C 180,E1 -12426.689,E2 -12426.689} C_VEL
LIN {X 0,Y 376.074,Z 222.636,A -85,B 0,C 180,E1 -12429.682,E2 -12429.682} C_VEL
LIN {X 0,Y 376.045,Z 222.64,A -85,B 0,C 180,E1 -12433.659,E2 -12433.659} C_VEL
LIN {X 0,Y 375.999,Z 222.645,A -85,B 0,C 180,E1 -12437.608,E2 -12437.608} C_VEL
LIN {X 0,Y 375.936,Z 222.658,A -85,B 0,C 180,E1 -12440.834,E2 -12440.834} C_VEL
LIN {X 0,Y 375.946,Z 222.654,A -85,B 0,C 180,E1 -12444.284,E2 -12444.284} C_VEL
LIN {X 0,Y 375.979,Z 222.654,A -85,B 0,C 180,E1 -12446.655,E2 -12446.655} C_VEL
LIN {X 0,Y 375.924,Z 222.659,A -85,B 0,C 180,E1 -12450.316,E2 -12450.316} C_VEL
LIN {X 0,Y 375.924,Z 222.657,A -85,B 0,C 180,E1 -12454.115,E2 -12454.115} C_VEL
LIN {X 0,Y 375.918,Z 222.659,A -85,B 0,C 180,E1 -12456.745,E2 -12456.745} C_VEL
LIN {X 0,Y 375.953,Z 222.653,A -85,B 0,C 180,E1 -12459.973,E2 -12459.973} C_VEL
LIN {X 0,Y 375.9,Z 222.659,A -85,B 0,C 180,E1 -12463.77,E2 -12463.77} C_VEL
LIN {X 0,Y 375.907,Z 222.658,A -85,B 0,C 180,E1 -12466.815,E2 -12466.815} C_VEL
LIN {X 0,Y 375.939,Z 222.656,A -85,B 0,C 180,E1 -12470.541,E2 -12470.541} C_VEL
LIN {X 0,Y 375.942,Z 222.653,A -85,B 0,C 180,E1 -12473.5,E2 -12473.5} C_VEL
LIN {X 0,Y 375.941,Z 222.657,A -85,B 0,C 180,E1 -12475.892,E2 -12475.892} C_VEL
LIN {X 0,Y 375.947,Z 222.654,A -85,B 0,C 180,E1 -12479.691,E2 -12479.691} C_VEL
LIN {X 0,Y 376.005,Z 222.645,A -85,B 0,C 180,E1 -12483.352,E2 -12483.352} C_VEL
LIN {X 0,Y 375.967,Z 222.649,A -85,B 0,C 180,E1 -12486.891,E2 -12486.891} C_VEL
LIN {X 0,Y 375.987,Z 222.649,A -85,B 0,C 180,E1 -12490.343,E2 -12490.343} C_VEL
LIN {X 0,Y 376.018,Z 222.649,A -85,B 0,C 180,E1 -12493.722,E2 -12493.722} C_VEL
LIN {X 0,Y 376.097,Z 222.634,A -85,B 0,C 180,E1 -12497.045,E2 -12497.045} C_VEL
LIN {X 0,Y 376.109,Z 222.633,A -85,B 0,C 180,E1 -12500.321,E2 -12500.321} C_VEL
LIN {X 0,Y 376.229,Z 222.769,A -85,B 0,C 180,E1 -12502.759,E2 -12502.759} C_VEL
LIN {X 0,Y 377.479,Z 229.874,A -85,B 0,C 180,E1 -12504.544,E2 -12504.544} C_VEL
LIN {X 0,Y 379.791,Z 238.207,A -85,B 0,C 180,E1 -12504.822,E2 -12504.822} C_VEL
LIN {X 0,Y 382.568,Z 253.318,A -85,B 0,C 180,E1 -12505.244,E2 -12505.244} C_VEL
LIN {X 0,Y 381.253,Z 336.956,A -85,B 0,C 180,E1 -12506.832,E2 -12506.832} C_VEL
LIN {X 0,Y 380.861,Z 350.164,A -85,B 0,C 180,E1 -12507.292,E2 -12507.292} C_VEL
LIN {X 0,Y 380.294,Z 363.036,A -85,B 0,C 180,E1 -12507.961,E2 -12507.961} C_VEL
LIN {X 0,Y 379.675,Z 374.399,A -85,B 0,C 180,E1 -12508.763,E2 -12508.763} C_VEL
LIN {X 0,Y 378.78,Z 386.466,A -85,B 0,C 180,E1 -12509.869,E2 -12509.869} C_VEL
LIN {X 0,Y 377.917,Z 396.845,A -85,B 0,C 180,E1 -12511.067,E2 -12511.067} C_VEL
LIN {X 0,Y 377.143,Z 406.162,A -85,B 0,C 180,E1 -12512.405,E2 -12512.405} C_VEL
LIN {X 0,Y 376.35,Z 415.187,A -85,B 0,C 180,E1 -12514.017,E2 -12514.017} C_VEL
LIN {X 0,Y 375.7,Z 422.469,A -85,B 0,C 180,E1 -12515.637,E2 -12515.637} C_VEL
LIN {X 0,Y 375.374,Z 427.792,A -85,B 0,C 180,E1 -12517.117,E2 -12517.117} C_VEL
LIN {X 0,Y 375.023,Z 432.152,A -85,B 0,C 180,E1 -12518.623,E2 -12518.623} C_VEL
LIN {X 0,Y 374.751,Z 435.814,A -85,B 0,C 180,E1 -12520.264,E2 -12520.264} C_VEL
LIN {X 0,Y 374.598,Z 438.443,A -85,B 0,C 180,E1 -12521.911,E2 -12521.911} C_VEL
LIN {X 0,Y 374.508,Z 439.68,A -85,B 0,C 180,E1 -12523.015,E2 -12523.015} C_VEL
LIN {X 0,Y 374.447,Z 440.471,A -85,B 0,C 180,E1 -12524.166,E2 -12524.166} C_VEL
LIN {X 0,Y 373.737,Z 440.839,A -85,B 0,C 180,E1 -12525.063,E2 -12525.063} C_VEL
LIN {X 0,Y 370.888,Z 440.942,A -85,B 0,C 180,E1 -12526.525,E2 -12526.525} C_VEL
LIN {X 0,Y 368.565,Z 440.513,A -85,B 0,C 180,E1 -12527.705,E2 -12527.705} C_VEL
LIN {X 0,Y 367.653,Z 439.857,A -85,B 0,C 180,E1 -12528.613,E2 -12528.613} C_VEL
LIN {X 0,Y 367.622,Z 439.55,A -85,B 0,C 180,E1 -12528.919,E2 -12528.919} C_VEL
LIN {X 0,Y 367.954,Z 437.288,A -85,B 0,C 180,E1 -12530.625,E2 -12530.625} C_VEL
LIN {X 0,Y 368.373,Z 433.772,A -85,B 0,C 180,E1 -12532.431,E2 -12532.431} C_VEL
LIN {X 0,Y 368.993,Z 429.113,A -85,B 0,C 180,E1 -12534.193,E2 -12534.193} C_VEL
LIN {X 0,Y 369.814,Z 423.201,A -85,B 0,C 180,E1 -12535.918,E2 -12535.918} C_VEL
LIN {X 0,Y 370.822,Z 415.576,A -85,B 0,C 180,E1 -12537.667,E2 -12537.667} C_VEL
LIN {X 0,Y 371.864,Z 407.71,A -85,B 0,C 180,E1 -12539.12,E2 -12539.12} C_VEL
LIN {X 0,Y 373.021,Z 398.035,A -85,B 0,C 180,E1 -12540.576,E2 -12540.576} C_VEL
LIN {X 0,Y 374.127,Z 388.451,A -85,B 0,C 180,E1 -12541.733,E2 -12541.733} C_VEL
LIN {X 0,Y 375.394,Z 376.453,A -85,B 0,C 180,E1 -12542.882,E2 -12542.882} C_VEL
LIN {X 0,Y 376.345,Z 364.827,A -85,B 0,C 180,E1 -12543.748,E2 -12543.748} C_VEL
LIN {X 0,Y 377.09,Z 352.639,A -85,B 0,C 180,E1 -12544.42,E2 -12544.42} C_VEL
LIN {X 0,Y 377.618,Z 338.847,A -85,B 0,C 180,E1 -12544.936,E2 -12544.936} C_VEL
LIN {X 0,Y 379.115,Z 269.941,A -85,B 0,C 180,E1 -12546.295,E2 -12546.295} C_VEL
LIN {X 0,Y 379.291,Z 254.469,A -85,B 0,C 180,E1 -12546.604,E2 -12546.604} C_VEL
LIN {X 0,Y 377.205,Z 246.341,A -85,B 0,C 180,E1 -12546.926,E2 -12546.926} C_VEL
LIN {X 0,Y 370.565,Z 230.726,A -85,B 0,C 180,E1 -12547.788,E2 -12547.788} C_VEL
LIN {X 0,Y 368.961,Z 223.529,A -85,B 0,C 180,E1 -12549.827,E2 -12549.827} C_VEL
LIN {X 0,Y 368.963,Z 223.528,A -85,B 0,C 180,E1 -12553.629,E2 -12553.629} C_VEL
LIN {X 0,Y 368.941,Z 223.529,A -85,B 0,C 180,E1 -12556.704,E2 -12556.704} C_VEL
LIN {X 0,Y 368.941,Z 223.527,A -85,B 0,C 180,E1 -12559.634,E2 -12559.634} C_VEL
LIN {X 0,Y 368.888,Z 223.532,A -85,B 0,C 180,E1 -12563.143,E2 -12563.143} C_VEL
LIN {X 0,Y 368.881,Z 223.535,A -85,B 0,C 180,E1 -12566.461,E2 -12566.461} C_VEL
LIN {X 0,Y 368.914,Z 223.526,A -85,B 0,C 180,E1 -12569.045,E2 -12569.045} C_VEL
LIN {X 0,Y 368.963,Z 223.519,A -85,B 0,C 180,E1 -12571.563,E2 -12571.563} C_VEL
LIN {X 0,Y 368.94,Z 223.519,A -85,B 0,C 180,E1 -12575.224,E2 -12575.224} C_VEL
LIN {X 0,Y 368.952,Z 223.517,A -85,B 0,C 180,E1 -12578.959,E2 -12578.959} C_VEL
LIN {X 0,Y 368.971,Z 223.517,A -85,B 0,C 180,E1 -12582.257,E2 -12582.257} C_VEL
LIN {X 0,Y 369.016,Z 223.515,A -85,B 0,C 180,E1 -12586.228,E2 -12586.228} C_VEL
LIN {X 0,Y 369.043,Z 223.513,A -85,B 0,C 180,E1 -12590.131,E2 -12590.131} C_VEL
LIN {X 0,Y 369.18,Z 223.496,A -85,B 0,C 180,E1 -12593.442,E2 -12593.442} C_VEL
LIN {X 0,Y 369.29,Z 223.48,A -85,B 0,C 180,E1 -12597.819,E2 -12597.819} C_VEL
LIN {X 0,Y 369.431,Z 223.458,A -85,B 0,C 180,E1 -12600,E2 -12600} C_VEL
LIN {X 0,Y 369.29,Z 223.475,A -85,B 0,C 180,E1 -12602.182,E2 -12602.182} C_VEL
LIN {X 0,Y 369.153,Z 223.49,A -85,B 0,C 180,E1 -12606.559,E2 -12606.559} C_VEL
LIN {X 0,Y 369.043,Z 223.502,A -85,B 0,C 180,E1 -12609.869,E2 -12609.869} C_VEL
LIN {X 0,Y 369.017,Z 223.51,A -85,B 0,C 180,E1 -12613.773,E2 -12613.773} C_VEL
LIN {X 0,Y 368.973,Z 223.519,A -85,B 0,C 180,E1 -12617.744,E2 -12617.744} C_VEL
LIN {X 0,Y 368.891,Z 223.533,A -85,B 0,C 180,E1 -12621.222,E2 -12621.222} C_VEL
LIN {X 0,Y 368.906,Z 223.533,A -85,B 0,C 180,E1 -12624.779,E2 -12624.779} C_VEL
LIN {X 0,Y 368.896,Z 223.531,A -85,B 0,C 180,E1 -12628.444,E2 -12628.444} C_VEL
LIN {X 0,Y 368.875,Z 223.534,A -85,B 0,C 180,E1 -12632.241,E2 -12632.241} C_VEL
LIN {X 0,Y 368.909,Z 223.531,A -85,B 0,C 180,E1 -12635.001,E2 -12635.001} C_VEL
LIN {X 0,Y 368.868,Z 223.539,A -85,B 0,C 180,E1 -12638.636,E2 -12638.636} C_VEL
LIN {X 0,Y 368.864,Z 223.523,A -85,B 0,C 180,E1 -12642.009,E2 -12642.009} C_VEL
LIN {X 0,Y 368.87,Z 223.534,A -85,B 0,C 180,E1 -12645.177,E2 -12645.177} C_VEL
LIN {X 0,Y 368.864,Z 223.539,A -85,B 0,C 180,E1 -12648.177,E2 -12648.177} C_VEL
LIN {X 0,Y 368.872,Z 223.537,A -85,B 0,C 180,E1 -12651.368,E2 -12651.368} C_VEL
LIN {X 0,Y 368.933,Z 223.529,A -85,B 0,C 180,E1 -12655.148,E2 -12655.148} C_VEL
LIN {X 0,Y 368.937,Z 223.628,A -85,B 0,C 180,E1 -12658.49,E2 -12658.49} C_VEL
LIN {X 0,Y 371.686,Z 235.204,A -85,B 0,C 180,E1 -12661.5,E2 -12661.5} C_VEL
LIN {X 0,Y 373.721,Z 245.683,A -85,B 0,C 180,E1 -12664.073,E2 -12664.073} C_VEL
LIN {X 0,Y 372.422,Z 258.936,A -85,B 0,C 180,E1 -12666.947,E2 -12666.947} C_VEL
LIN {X 0,Y 372.195,Z 261.116,A -85,B 0,C 180,E1 -12667.415,E2 -12667.415} C_VEL
LIN {X 0,Y 376.625,Z 283.768,A -85,B 0,C 180,E1 -12668.226,E2 -12668.226} C_VEL
LIN {X 0,Y 378.626,Z 297.76,A -85,B 0,C 180,E1 -12668.659,E2 -12668.659} C_VEL
LIN {X 0,Y 377.23,Z 370.206,A -85,B 0,C 180,E1 -12670.087,E2 -12670.087} C_VEL
LIN {X 0,Y 376.552,Z 383.305,A -85,B 0,C 180,E1 -12670.547,E2 -12670.547} C_VEL
LIN {X 0,Y 375.526,Z 395.4,A -85,B 0,C 180,E1 -12671.165,E2 -12671.165} C_VEL
LIN {X 0,Y 374.451,Z 406.82,A -85,B 0,C 180,E1 -12671.959,E2 -12671.959} C_VEL
LIN {X 0,Y 373.289,Z 417.289,A -85,B 0,C 180,E1 -12672.892,E2 -12672.892} C_VEL
LIN {X 0,Y 372.065,Z 428.06,A -85,B 0,C 180,E1 -12674.103,E2 -12674.103} C_VEL
LIN {X 0,Y 370.881,Z 437.694,A -85,B 0,C 180,E1 -12675.445,E2 -12675.445} C_VEL
LIN {X 0,Y 369.965,Z 445.763,A -85,B 0,C 180,E1 -12676.822,E2 -12676.822} C_VEL
LIN {X 0,Y 368.912,Z 453.627,A -85,B 0,C 180,E1 -12678.46,E2 -12678.46} C_VEL
LIN {X 0,Y 368.257,Z 459.936,A -85,B 0,C 180,E1 -12680.109,E2 -12680.109} C_VEL
LIN {X 0,Y 367.802,Z 464.981,A -85,B 0,C 180,E1 -12681.759,E2 -12681.759} C_VEL
LIN {X 0,Y 367.556,Z 468.909,A -85,B 0,C 180,E1 -12683.411,E2 -12683.411} C_VEL
LIN {X 0,Y 367.454,Z 472.565,A -85,B 0,C 180,E1 -12685.611,E2 -12685.611} C_VEL
LIN {X 0,Y 367.404,Z 473.781,A -85,B 0,C 180,E1 -12686.709,E2 -12686.709} C_VEL
LIN {X 0,Y 367.451,Z 474.559,A -85,B 0,C 180,E1 -12687.806,E2 -12687.806} C_VEL
LIN {X 0,Y 367.539,Z 474.944,A -85,B 0,C 180,E1 -12688.903,E2 -12688.903} C_VEL
LIN {X 0,Y 367.545,Z 474.94,A -85,B 0,C 180,E1 -12689.998,E2 -12689.998} C_VEL
LIN {X 0,Y 367.56,Z 474.545,A -85,B 0,C 180,E1 -12691.094,E2 -12691.094} C_VEL
LIN {X 0,Y 367.49,Z 473.708,A -85,B 0,C 180,E1 -12692.19,E2 -12692.19} C_VEL
LIN {X 0,Y 367.506,Z 470.802,A -85,B 0,C 180,E1 -12694.385,E2 -12694.385} C_VEL
LIN {X 0,Y 367.522,Z 467.357,A -85,B 0,C 180,E1 -12696.075,E2 -12696.075} C_VEL
LIN {X 0,Y 367.681,Z 463.004,A -85,B 0,C 180,E1 -12697.687,E2 -12697.687} C_VEL
LIN {X 0,Y 367.968,Z 457.337,A -85,B 0,C 180,E1 -12699.34,E2 -12699.34} C_VEL
LIN {X 0,Y 368.44,Z 450.237,A -85,B 0,C 180,E1 -12700.994,E2 -12700.994} C_VEL
LIN {X 0,Y 369.247,Z 441.348,A -85,B 0,C 180,E1 -12702.64,E2 -12702.64} C_VEL
LIN {X 0,Y 370.122,Z 431.23,A -85,B 0,C 180,E1 -12704.148,E2 -12704.148} C_VEL
LIN {X 0,Y 370.937,Z 420.862,A -85,B 0,C 180,E1 -12705.379,E2 -12705.379} C_VEL
LIN {X 0,Y 371.855,Z 409.361,A -85,B 0,C 180,E1 -12706.466,E2 -12706.466} C_VEL
LIN {X 0,Y 372.744,Z 397.384,A -85,B 0,C 180,E1 -12707.342,E2 -12707.342} C_VEL
LIN {X 0,Y 373.529,Z 384.861,A -85,B 0,C 180,E1 -12708.012,E2 -12708.012} C_VEL
LIN {X 0,Y 374.117,Z 372.023,A -85,B 0,C 180,E1 -12708.478,E2 -12708.478} C_VEL
LIN {X 0,Y 374.783,Z 333.47,A -85,B 0,C 180,E1 -12709.25,E2 -12709.25} C_VEL
LIN {X 0,Y 375.097,Z 295.131,A -85,B 0,C 180,E1 -12709.993,E2 -12709.993} C_VEL
LIN {X 0,Y 370.631,Z 261.944,A -85,B 0,C 180,E1 -12710.864,E2 -12710.864} C_VEL
LIN {X 0,Y 372.135,Z 243.011,A -85,B 0,C 180,E1 -12714.84,E2 -12714.84} C_VEL
LIN {X 0,Y 371.969,Z 238.821,A -85,B 0,C 180,E1 -12715.753,E2 -12715.753} C_VEL
LIN {X 0,Y 369.824,Z 227.471,A -85,B 0,C 180,E1 -12718.36,E2 -12718.36} C_VEL
LIN {X 0,Y 368.952,Z 223.529,A -85,B 0,C 180,E1 -12719.338,E2 -12719.338} C_VEL
LIN {X 0,Y 368.882,Z 223.532,A -85,B 0,C 180,E1 -12723.039,E2 -12723.039} C_VEL
LIN {X 0,Y 368.899,Z 223.534,A -85,B 0,C 180,E1 -12726.193,E2 -12726.193} C_VEL
LIN {X 0,Y 368.882,Z 223.532,A -85,B 0,C 180,E1 -12728.949,E2 -12728.949} C_VEL
LIN {X 0,Y 368.859,Z 223.54,A -85,B 0,C 180,E1 -12732.005,E2 -12732.005} C_VEL
LIN {X 0,Y 368.926,Z 223.527,A -85,B 0,C 180,E1 -12735.182,E2 -12735.182} C_VEL
LIN {X 0,Y 368.918,Z 223.53,A -85,B 0,C 180,E1 -12738.182,E2 -12738.182} C_VEL
LIN {X 0,Y 368.883,Z 223.534,A -85,B 0,C 180,E1 -12741.355,E2 -12741.355} C_VEL
LIN {X 0,Y 368.904,Z 223.531,A -85,B 0,C 180,E1 -12745.143,E2 -12745.143} C_VEL
LIN {X 0,Y 368.895,Z 223.531,A -85,B 0,C 180,E1 -12749.043,E2 -12749.043} C_VEL
LIN {X 0,Y 368.944,Z 223.531,A -85,B 0,C 180,E1 -12751.561,E2 -12751.561} C_VEL
LIN {X 0,Y 368.922,Z 223.53,A -85,B 0,C 180,E1 -12755.222,E2 -12755.222} C_VEL
LIN {X 0,Y 368.932,Z 223.527,A -85,B 0,C 180,E1 -12758.957,E2 -12758.957} C_VEL
LIN {X 0,Y 368.949,Z 223.524,A -85,B 0,C 180,E1 -12762.255,E2 -12762.255} C_VEL
LIN {X 0,Y 368.994,Z 223.518,A -85,B 0,C 180,E1 -12766.226,E2 -12766.226} C_VEL
LIN {X 0,Y 369.028,Z 223.514,A -85,B 0,C 180,E1 -12770.13,E2 -12770.13} C_VEL
LIN {X 0,Y 369.156,Z 223.498,A -85,B 0,C 180,E1 -12772.341,E2 -12772.341} C_VEL
LIN {X 0,Y 369.106,Z 223.505,A -85,B 0,C 180,E1 -12774.537,E2 -12774.537} C_VEL
LIN {X 0,Y 369.269,Z 223.484,A -85,B 0,C 180,E1 -12777.818,E2 -12777.818} C_VEL
LIN {X 0,Y 369.41,Z 223.466,A -85,B 0,C 180,E1 -12780,E2 -12780} C_VEL
LIN {X 0,Y 369.267,Z 223.484,A -85,B 0,C 180,E1 -12782.181,E2 -12782.181} C_VEL
LIN {X 0,Y 369.138,Z 223.501,A -85,B 0,C 180,E1 -12786.675,E2 -12786.675} C_VEL
LIN {X 0,Y 369.023,Z 223.514,A -85,B 0,C 180,E1 -12789.869,E2 -12789.869} C_VEL
LIN {X 0,Y 368.993,Z 223.518,A -85,B 0,C 180,E1 -12793.773,E2 -12793.773} C_VEL
LIN {X 0,Y 368.959,Z 223.522,A -85,B 0,C 180,E1 -12797.77,E2 -12797.77} C_VEL
LIN {X 0,Y 368.867,Z 223.535,A -85,B 0,C 180,E1 -12801.223,E2 -12801.223} C_VEL
LIN {X 0,Y 368.913,Z 223.533,A -85,B 0,C 180,E1 -12804.778,E2 -12804.778} C_VEL
LIN {X 0,Y 368.922,Z 223.528,A -85,B 0,C 180,E1 -12807.206,E2 -12807.206} C_VEL
LIN {X 0,Y 368.874,Z 223.535,A -85,B 0,C 180,E1 -12810.99,E2 -12810.99} C_VEL
LIN {X 0,Y 368.901,Z 223.532,A -85,B 0,C 180,E1 -12814.857,E2 -12814.857} C_VEL
LIN {X 0,Y 368.871,Z 223.537,A -85,B 0,C 180,E1 -12818.643,E2 -12818.643} C_VEL
LIN {X 0,Y 368.85,Z 223.539,A -85,B 0,C 180,E1 -12822.013,E2 -12822.013} C_VEL
LIN {X 0,Y 368.85,Z 223.536,A -85,B 0,C 180,E1 -12825.179,E2 -12825.179} C_VEL
LIN {X 0,Y 368.857,Z 223.541,A -85,B 0,C 180,E1 -12828.181,E2 -12828.181} C_VEL
LIN {X 0,Y 368.885,Z 223.532,A -85,B 0,C 180,E1 -12831.364,E2 -12831.364} C_VEL
LIN {X 0,Y 368.916,Z 223.528,A -85,B 0,C 180,E1 -12835.15,E2 -12835.15} C_VEL
LIN {X 0,Y 368.913,Z 223.528,A -85,B 0,C 180,E1 -12839.05,E2 -12839.05} C_VEL
LIN {X 0,Y 368.949,Z 223.524,A -85,B 0,C 180,E1 -12842.8,E2 -12842.8} C_VEL
LIN {X 0,Y 368.921,Z 223.532,A -85,B 0,C 180,E1 -12846.121,E2 -12846.121} C_VEL
LIN {X 0,Y 368.926,Z 223.532,A -85,B 0,C 180,E1 -12849.95,E2 -12849.95} C_VEL
LIN {X 0,Y 368.96,Z 223.524,A -85,B 0,C 180,E1 -12853.402,E2 -12853.402} C_VEL
LIN {X 0,Y 369.052,Z 223.511,A -85,B 0,C 180,E1 -12856.793,E2 -12856.793} C_VEL
LIN {X 0,Y 369.059,Z 223.512,A -85,B 0,C 180,E1 -12860.134,E2 -12860.134} C_VEL
LIN {X 0,Y 369.15,Z 223.585,A -85,B 0,C 180,E1 -12862.516,E2 -12862.516} C_VEL
LIN {X 0,Y 370.414,Z 230.344,A -85,B 0,C 180,E1 -12864.217,E2 -12864.217} C_VEL
LIN {X 0,Y 373.262,Z 240.492,A -85,B 0,C 180,E1 -12864.559,E2 -12864.559} C_VEL
LIN {X 0,Y 375.769,Z 253.555,A -85,B 0,C 180,E1 -12864.937,E2 -12864.937} C_VEL
LIN {X 0,Y 374.398,Z 337.987,A -85,B 0,C 180,E1 -12866.577,E2 -12866.577} C_VEL
LIN {X 0,Y 373.948,Z 351.615,A -85,B 0,C 180,E1 -12867.073,E2 -12867.073} C_VEL
LIN {X 0,Y 373.39,Z 364.498,A -85,B 0,C 180,E1 -12867.777,E2 -12867.777} C_VEL
LIN {X 0,Y 372.689,Z 375.844,A -85,B 0,C 180,E1 -12868.616,E2 -12868.616} C_VEL
LIN {X 0,Y 371.781,Z 387.591,A -85,B 0,C 180,E1 -12869.731,E2 -12869.731} C_VEL
LIN {X 0,Y 370.921,Z 397.811,A -85,B 0,C 180,E1 -12870.952,E2 -12870.952} C_VEL
LIN {X 0,Y 370.035,Z 407.806,A -85,B 0,C 180,E1 -12872.451,E2 -12872.451} C_VEL
LIN {X 0,Y 369.251,Z 416.609,A -85,B 0,C 180,E1 -12874.094,E2 -12874.094} C_VEL
LIN {X 0,Y 368.593,Z 423.651,A -85,B 0,C 180,E1 -12875.746,E2 -12875.746} C_VEL
LIN {X 0,Y 368.301,Z 428.438,A -85,B 0,C 180,E1 -12877.128,E2 -12877.128} C_VEL
LIN {X 0,Y 367.919,Z 433.056,A -85,B 0,C 180,E1 -12878.791,E2 -12878.791} C_VEL
